// ---- Sequence/ST_SequenceInfo.TcDUT
{attribute 'enable_dynamic_creation'}
TYPE ST_SequenceInfo :
STRUCT
	nSequId 		: UDINT;			//4 Byte
	nStepNr 		: UINT;				//2 Byte
	eSequenceState	: E_SequenceState;	//1 Byte
	eStepState		: E_StepState;		//1 Byte
	nInfo			: DINT;				//4 Byte
END_STRUCT
END_TYPE

// ---- Sequence/ST_Step.TcDUT
{attribute 'enable_dynamic_creation'}
TYPE ST_Step :
STRUCT
	nStepNr				: UINT;	
	bStop				: BOOL;
	tDelay				: TIME;
	nTimerId			: USINT;
	eState 				: E_StepState;
	stActionData		: ST_ActionData;
	nActionId			: UINT;
	pCondi				: POINTER TO FB_CondiBase;
	aFollower			: ARRAY[0..9] OF UINT;
	bFollowerInQueue	: BOOL;	//Follwoer wurden in ProcessingQueue eingetragen
	bHasForerunner		: BOOL; //Hat einen Vorgänger (PreStep oder SpecStep) auf den gewartet wird
	bActionResultIsValid: BOOL;
	nActionResult		: DINT;
	nInfo				: DINT;
	bInfoChanged		: BOOL; //wird gesetzt, sobald sich der State oder nInfo ändert
END_STRUCT
END_TYPE

// ---- Configuration/GVL_ObjectArrays.TcGVL
{attribute 'contextName':='PlcTask'}
VAR_GLOBAL
	//Instanzierung der Objekte, sollten vom jeweiligem Objekttyp die Anzahl geändert werden müssen
	//dann die jeweilige Constante cMax....... ändern
	
	//MultiZ-Tools
	afbMzHead 			: ARRAY[1..cMaxMzHeads] OF FB_MzHead;				//MultiZ-Kopf - Anzahl bei 2 Ebenenplotter auf 2 Stück erhöhen
	afbPiezoPip 		: ARRAY[1..cMaxPiezoPips] OF FB_PiezoPip;			//Piezopipetten - Anzahl kann theoretisch auf 7 erhöht werden (pro Z-Scheibe 1 Pipette)
	afbPassivPip		: ARRAY[1..cMaxPassivPips] OF FB_PassivPip;			//Passivpipetten - Anzahl kann theoretisch auf 7 erhöht werden (pro Z-Scheibe 1 Pipette)
	afbPowderPip 		: ARRAY[1..cMaxPowderPips] OF FB_PowderPip;			//Pulverpipette
	afbMultiCartHolder	: ARRAY[1..cMaxMultiCartHolder] OF FB_MultiCartHolder;	//ehemals Corshell-Dispenser
	afbHybridDispenser	: ARRAY[1..cMaxHybridDispenser] OF FB_HybridDispenser;//
	afbCartDisp			: ARRAY[1..cMaxCartDisp] OF FB_CartDispenser;		//Kartuschen-Dispenser
	afbCartDispStirrer	: ARRAY[1..cMaxCartDispStirrer] OF FB_CartDispStirrer;	//Kartuschen-Dispenser mit Rührer
	afbCartHolder		: ARRAY[1..cMaxCartHolder] OF FB_CartHolder;		//Kartuschen-Halter
	afbCamera			: ARRAY[1..cMaxCameras] OF FB_Camera;				//Kamera oder Mikroskop oder Scanner
	afbZLevelSensor		: ARRAY[1..cMaxZLevelSensors] OF FB_ZLevelSensor;	//Z-Levelsensor
	afbStampSupport		: ARRAY[1..cMaxStampSupports] OF FB_StampSupport;	//Stempelkopf/Support
	afbDeloDot			: ARRAY[1..cMaxDeloDots] OF FB_DeloDot;				//DeloDot
	afbExposure			: ARRAY[1..cMaxExposure] OF FB_Exposure;			//Belichtung
	afbTriplePip		: ARRAY[1..cMaxTriplePip] OF FB_TriplePip;			//TriplePipette
	afbFlipTubeHandler	: ARRAY[1..cMaxFlipTubeHandler] OF FB_FlipTubeHandler;
	afbLuer				: ARRAY[1..cMaxLuer] OF FB_Luer;					
	afbVacuumHandler	: ARRAY[1..cMaxLuer] OF FB_VacuumHandler;
	afbSinglePiezoHolder: ARRAY[1..cMaxSinglePiezoHolder] OF FB_SingelPiezoHolder;
	afbTwinPiezoHolder	: ARRAY[1..cMaxTwinPiezoHolder] OF FB_TwinPiezoHolder;
	afbSolenoidPip		: ARRAY[1..cMaxSolenoidPip] OF FB_SolenoidPip;
	afbExtruder			: ARRAY[1..cMaxExtruder] OF FB_Extruder;
	afbpHElectrode		: ARRAY[1..cMaxpHElectrodes] OF FB_pHElectrode;
	afbTitrationTool	: ARRAY[1..cMaxTitrationTools] OF FB_TitrationTool;
	afbTwinExtruder		: ARRAY[1..cMaxTwinExtruder] OF FB_TwinExtruder;
	afbVermesDisp		: ARRAY[1..cMaxVermesDisp] OF FB_VermesDisp;
	afbDummyTool		: ARRAY[1..cMaxDummyTools] OF FB_DummyTool;	//Universelles Tool, welches außer den Move-Actions keine speziellen Funktionalitäten hat
	afbGripper			: ARRAY[1..cMaxGripper] OF FB_Gripper;
	afbPickPlacePip		: ARRAY[1..cMaxPickPlacePip] OF FB_PickPlacePip;
	
	//passive Targets
	afbWorkplate		: ARRAY[1..cMaxWorkplates] OF FB_Workplate;			//repräsentiert die gesamte Arbeitsfläche (Root) und kann nur 1x vorhanden sein
	afbSpotArray		: ARRAY[1..cMaxSpotArrays] OF FB_SpotArray;			//SpotArray
	afbDryPad			: ARRAY[1..cMaxDrayPads] OF FB_DryPad;				//Trockenpad
	afbSeptumWaste		: ARRAY[1..cMaxSeptumWaste] OF FB_SeptumWaste;		//SeptumWaste
	
	afbStampMagazine	: ARRAY[1..cMaxStampMagazines] OF FB_StampMagazine;	//Stempelmagazin
	afbSpotPattern		: ARRAY[1..cMaxSpotPatterns] OF FB_SpotPattern;		//Spotpattern
	afbNeedleRack		: ARRAY[1..cMaxNeedleRack] OF FB_NeedleRack;		//NeedleRack
	afbTipRack			: ARRAY[1..cMaxTipRack] OF FB_TipRack;				//TipRack
	afbFlipTubeRack		: ARRAY[1..cMaxFlipTubeRack] OF FB_FlipTubeRack;	//FlipTubeRack
	afbSeptumRack		: ARRAY[1..cMaxSeptumRack] OF FB_SeptumRack;		//SeptumRack
	afbVialRack			: ARRAY[1..cMaxVialRack] OF FB_VialRack;			//VialRack
	afbPortRack			: ARRAY[1..cMaxPortRack] OF FB_PortRack;			//PortRack
	afbpHElectrodeCapRack : ARRAY[1..cMaxpHElectrodeCapRack] OF FB_pHElectrodeCapRack;	//Rack für Konditionierungsgefäß pH-Elektrode
	afbTipCleanerGen2	: ARRAY[1..cMaxTipCleanerGen2] OF FB_TipCleanerGen2;
	
	//aktive Targets
	afbWashStation		: ARRAY[1..cMaxWashStations] OF FB_WashStation;		//Waschstation
	afbTipCleaner		: ARRAY[1..cMaxTipCleaners] OF FB_TipCleaner;		//Tip-Reinigung
	afbTipCalibrator	: ARRAY[1..cMaxTipCalibrators] OF FB_TipCalibrator;	//Tip-Kalibrierung
	afbStroboscope		: ARRAY[1..cMaxStroboscopes] OF FB_Stroboscope;		//Stroboskop
	afbMtpHolder		: ARRAY[1..cMaxMtpHolders] OF FB_MtpHolder;			//Mikrotiterplattenhalter, kann heizen oder kühlen
	afbSubstHolder		: ARRAY[1..cMaxSubstHolders] OF FB_SubstHolder;		//Substrathalter, kann heizen oder kühlen
	{IF defined(Unistat)}
	afbSubstHolderUnistat: ARRAY[1..cMaxSubstHolderUnistat] OF FB_SubstHolderUnistat;		//Substrathalter mit Huber Unistat 405
	{END_IF}
	afbInkStation		: ARRAY[1..cMaxInkStations] OF FB_InkStation;		//Lackschleuder für µCP
	afbPowderStation	: ARRAY[1..cMaxPowderStations] OF FB_PowderStation;	//Pulvervorrat für Pulverpipette
	afbReactor			: ARRAY[1..cMaxReactors] OF FB_Reactor;				//Reaktor
	afbLiquidReserve	: ARRAY[1..cMaxLiquidReserve] OF FB_LiquidReserve;	//LiquidReserve
	afbHighVoltTray		: ARRAY[1..cMaxHighVoltTray] OF FB_HighVoltTray;	//Hochspannungstablett für MES
	afbWorkplateCamera	: ARRAY[1..cMaxWorkplateCameras] OF FB_WorkplateCamera;
	afbCustomUnitType1	: ARRAY[1..cMaxCustomUnitTyp1] OF FB_CustomUnitType1;
	afbCustomUnitType2	: ARRAY[1..cMaxCustomUnitTyp2] OF FB_CustomUnitType2;
	afbTrayTransporter	: ARRAY[1..cMaxTrayTransporter] OF FB_TrayTransporter;
	
	//sonstige Devices
	afbDiluter			: ARRAY[1..cMaxDiluters] OF FB_Diluter;				//Spritzenpumpen
	afbDiluter3Inputs	: ARRAY[1..cMaxDiluters3Inputs] OF FB_Diluter3Inputs;
	afbStacker			: ARRAY[1..cMaxStacker] OF FB_Stacker;
	

	////////////////////////////////////////////////////////////////////////////////////////////////////////////////////////////////////////	
END_VAR

// ---- Configuration/GVL_ObjectConstants.TcGVL
VAR_GLOBAL CONSTANT
	//Legt die Anzahl der Instanzen der verschiedenen Objekt-Fbs fest.
	//Begrenzt die maximale Anzahl konfigurierbarer Objekt-Typen. 
	//MultiZ-Tools
	{IF defined (TwoHeads)}
	cMaxMzHeads			: USINT := 2;
	{ELSE}
	cMaxMzHeads			: USINT := 1;
	{END_IF}
	cMaxPickPlacePip	: UINT := 2;
	cMaxPiezoPips		: UINT := 4;
	cMaxPassivPips		: UINT := 8;
	cMaxPowderPips		: UINT := 1;
	cMaxMultiCartHolder	: UINT := 1;
	cMaxHybridDispenser	: UINT := 1;
	cMaxCartDisp		: UINT := 4;
	cMaxCartDispStirrer	: UINT := 1;
	cMaxCartHolder		: UINT := 6;
	cMaxCameras			: UINT := 6;
	cMaxZLevelSensors	: UINT := 2;
	cMaxStampSupports	: UINT := 1;
	cMaxDeloDots		: UINT := 1;
	cMaxExposure		: UINT := 4;
	cMaxTriplePip		: UINT := 2;
	cMaxFlipTubeHandler	: UINT := 1;
	cMaxLuer			: UINT := 6;
	cMaxVacuumHandler	: UINT := 2;
	cMaxSinglePiezoHolder: UINT := 4;
	cMaxTwinPiezoHolder	: UINT := 1;
	cMaxSolenoidPip		: UINT := 1;
	cMaxExtruder		: UINT := 4;
	cMaxpHElectrodes	: UINT := 1;
	cMaxTitrationTools	: UINT := 3;
	cMaxTwinExtruder	: UINT := 1;
	cMaxVermesDisp		: UINT := 1;
	cMaxDummyTools		: UINT := 7;
	cMaxGripper			: UINT := 1;
	
	//passive Targets
	cMaxWorkplates		: UINT := 1;
	cMaxSpotArrays		: UINT := 50;
	cMaxDrayPads		: UINT := 3;
	cMaxStampMagazines	: UINT := 1;
	cMaxSpotPatterns	: UINT := 10;
	cMaxSeptumWaste		: UINT := 1;
	cMaxNeedleRack		: UINT := 3;
	cMaxTipRack			: UINT := 2;
	cMaxFlipTubeRack	: UINT := 3;
	cMaxSeptumRack		: UINT := 1;
	cMaxVialRack		: UINT := 3;
	cMaxPortRack		: UINT := 1;
	cMaxpHElectrodeCapRack: UINT := 1;
	cMaxTipCleanerGen2	: UINT := 2;
	
	//aktive Targets
	cMaxWashStations	: UINT := 2;
	cMaxTipCleaners		: UINT := 1;
	cMaxTipCalibrators	: UINT := 1;
	cMaxStroboscopes	: UINT := 1;
	cMaxMtpHolders		: UINT := 3;
	cMaxSubstHolders	: UINT := 2;
	cMaxSubstHolderUnistat	: UINT := 1;
	cMaxInkStations		: UINT := 1;
	cMaxPowderStations	: UINT := 1;
	cMaxReactors		: UINT := 1;
	cMaxLiquidReserve	: UINT := 1;
	cMaxHighVoltTray	: UINT := 1;
	cMaxWorkplateCameras: UINT := 1;
	cMaxCustomUnitTyp1	: UINT := 2;
	cMaxCustomUnitTyp2	: UINT := 1;
	cMaxTrayTransporter : UINT := 1;
	
	//sonstige Devices
	cMaxDiluters		: UINT := 8;
	cMaxDiluters3Inputs	: UINT := 2;
	cMaxStacker			: UINT := 1;
	
	//!!!!!!!!!!!!!!!!!!!!!!!!!!!!!!!!!!!!!!!!!!!!!!!!!!!!!!!!!!!!!!!!!!!!!!!!!!!!!!!!!!!!!!!!!!!!!!!
	//Achtung, unbedingt cMaxObjects anpassen - muss "mindestens" die Summe aller cMax..... ergeben
	cMaxObjects			: UINT := 1000;
	
	//Achtung, unbedingt cMaxDevices anpassen - muss "mindestens" die Summe aller cMax.....  
	//von MultiZ-Tools + aktive Targets + sonstige Devices ergeben 
	cMaxDevices			: UINT := 30;

END_VAR

// ---- Configuration/GVL_ObjMgmt.TcGVL
VAR_GLOBAL
	fbConfiguration		: FB_Configuration;
	fbObjectDirectory 	: FB_ObjectDirectory;
	nObjPropChangeCnt	: USINT;
END_VAR

// ---- GVLs/GVL_Hardware.TcGVL
{attribute 'contextName':='PlcTask'}
VAR_GLOBAL CONSTANT
	//Definition der Hardwarecomponenten
	{define MtpHeater}
	{IF defined(MtpHeater)}
	cNoOfMtpHeaters	: USINT := 1;
	cNodeIdMtpHeater1 : USINT := 10;
	{END_IF}
	
	{define SubstHeater}
	{IF defined(SubstHeater)}
	cNoOfSubstHeaters : USINT := 1;
	cNodeIdSubstHeater1 : USINT := 12;
	{END_IF}

	//{define Reactor}
	{IF defined(Reactor)}
	cNoOfReactDrives : USINT := 1;
	cNodeIdReactDrive1	: USINT := 4;
	cNoOfReactHeaters : USINT := 1;
	cNodeIdReactHeater1	: USINT := 5;
	{END_IF}
	
	//{define BottleRack}
	{IF defined(BottleRack)}
	cNoOfBottleRacks : USINT := 1;
	cNodeIdBottleRack1 : USINT := 20;
	{END_IF}
	
	{define IOExpander}
	{IF defined(IOExpander)}
	cNoOfIOExpanders : USINT := 1;
	cNodeIdIOExpander1 : USINT := 16;
	{END_IF}
	
	//{define TripleTrigger}
	{IF defined(TripleTrigger)}
	cNoOfTripleTriggers : USINT := 1;
	cNodeIdTripleTrigger1 : USINT := 14;
	{END_IF}
	
	//{define PowderStation}
	{IF defined(PowderStation)}
	cNoOfPowderStations : USINT := 1;
	cNodeIdPowderStation1 : USINT := 24;
	{END_IF}
	
	//{define InkStation}
	{IF defined(InkStation)}
	cNoOfInkStatSpinDrives 		: USINT := 1;
	cNodeIdInkStatSpinDrive1	: USINT := 32;
	cNoOfInkStatCoverDrives 	: USINT := 1;
	cNodeIdInkStatCoverDrive1	: USINT := 33;
	{END_IF}
	
	{define MultiPurpIO}
	{IF defined(MultiPurpIO)}
	cNoOfMultiPurpIO			: USINT := 1;
	cNodeIdMultiPurpIO			: USINT := 25;
	{END_IF}
	
	cNoOfLiquidBottles 	: USINT := 1;
	cNoOfWasteBottles 	: USINT := 1;
	cNoOfPneuChannels	: USINT := 4;
	cNoOfPumps			: USINT := 9; //höchste Pumpennummer
	cNoOfGearPumps		: USINT := 4; //hochste Nummer Zahnradpumpen
	cNoOfValves			: USINT := 14;//höchste Ventilnummer
	cNoOfDiluters		: USINT	:= 8;
	
	cLiquidBottleNrPCV	: USINT := 1;
	
END_VAR

VAR_GLOBAL
	
	stPlcInfo			: ST_PlcInfo;	//Information über Seriennummer und Versionen der Plc
	
	//CAN-Nodes
	aCanNodes				: ARRAY[1..126] OF BOOL;
	
	//Settings
	fbSettings 				: FB_Settings;
	
	fbCANOpenHwModuleList	: FB_HwModuleList;	//alle GeSim CANopen-Module
	
	//Diluter	
	aFbDiluterRef			: ARRAY[1..cNoOfDiluters] OF FB_HwRefDiluter;
	
	//MultiZ-Module
	aFbMultiZRef			: ARRAY[1..cMaxMzHeads] OF FB_MultiZRef;	//Gerätereferenz zu MultiZ 1 (2)
	fbMultiZRefList			: FB_HwModuleList;
	
	{IF defined(MtpHeater)}
	aFbMtpHeatRef			: ARRAY[1..cNoOfMtpHeaters] OF FB_HwRef4ChHeater;
	{END_IF}
	
	{IF defined(SubstHeater)}
	aFbSubstHeatRef			: ARRAY[1..cNoOfSubstHeaters] OF FB_HwRef4ChHeater;
	{END_IF}	

	{IF defined(Reactor)}
	aFbReactDriveRef		: ARRAY[1..cNoOfReactDrives] OF FB_HwRefReactDrive;
	aFbReactHeatRef			: ARRAY[1..cNoOfReactHeaters] OF FB_HwRefReactHeater;
	{END_IF}
	
	{IF defined(BottleRack)}
	aFbBottleRackRef		: ARRAY[1..cNoOfBottleRacks] OF FB_HwRefBottleRack;
	{END_IF}
	
	{IF defined(IOExpander)}
	aFbIOExpanderRef		: ARRAY[1..cNoOfIOExpanders] OF FB_HwRefIOExpander;
	{END_IF}
	
	{IF defined(TripleTrigger)}
	aFbTripleTriggerRef		: ARRAY[1..cNoOfTripleTriggers] OF FB_HwRefTripleTrigger;
	{END_IF}
	
	{IF defined(PowderStation)}
	aFbPowderStatRef		: ARRAY[1..cNoOfPowderStations] OF FB_HwRefPowderStat;
	{END_IF}
	
	{IF defined(InkStation)}
	aFbInkStatDrvSpinRef	: ARRAY[1..cNoOfInkStatSpinDrives] OF FB_HwRefInkStatDriveSpin;
	aFbInkStatDrvCoverRef	: ARRAY[1..cNoOfInkStatCoverDrives] OF FB_HwRefInkStatDriveCover;
	{END_IF}
	
	//Muss in Compilerdefinitionen definiert werden
	{IF defined(TrayTransporterL)}
	fbHwRefTrayLock			: FB_HwRefTrayLock;
	fbHwRefTrayTransSlider 	: FB_HwRefNanotecPD;
	fbHwRefDrivingPinLeft	: FB_HwRefTMCM1140(bSetDigiOut0:= FALSE, bSetDigiOut1:= TRUE,
											eLimitSwitchLeftConfig := E_TMCM_SwitchConfig.Deactivated,
											eLimitSwitchRightConfig := E_TMCM_SwitchConfig.Deactivated,
											eHomeSwitchConfig := E_TMCM_SwitchConfig.Inverted,
											eHomingMethode := E_TMCM_HomingMethode.SearchNegHomeSwitch,
											nMicrostepResol := 64, nPulseDivisor := 2, nFullStepRevo := 200);
	{ELSIF defined(TrayTransporterR)}
	fbHwRefTrayLock			: FB_HwRefTrayLock;
	fbHwRefTrayTransSlider 	: FB_HwRefNanotecPD;
	fbHwRefDrivingPinRight	: FB_HwRefTMCM1140(bSetDigiOut0:= FALSE, bSetDigiOut1:= TRUE,
											eLimitSwitchLeftConfig := E_TMCM_SwitchConfig.Deactivated,
											eLimitSwitchRightConfig := E_TMCM_SwitchConfig.Deactivated,
											eHomeSwitchConfig := E_TMCM_SwitchConfig.Inverted,
											eHomingMethode := E_TMCM_HomingMethode.SearchNegHomeSwitch,
											nMicrostepResol := 64, nPulseDivisor := 2, nFullStepRevo := 200);
	{ELSIF defined(TrayTransporterLR)}
	fbHwRefTrayLock			: FB_HwRefTrayLock;
	fbHwRefTrayTransSlider  : FB_HwRefNanotecPD;
	fbHwRefDrivingPinLeft	: FB_HwRefTMCM1140(bSetDigiOut0:= FALSE, bSetDigiOut1:= TRUE,
											eLimitSwitchLeftConfig := E_TMCM_SwitchConfig.Deactivated,
											eLimitSwitchRightConfig := E_TMCM_SwitchConfig.Deactivated,
											eHomeSwitchConfig := E_TMCM_SwitchConfig.Inverted,
											eHomingMethode := E_TMCM_HomingMethode.SearchNegHomeSwitch,
											nMicrostepResol := 64, nPulseDivisor := 2, nFullStepRevo := 200);
	fbHwRefDrivingPinRight	: FB_HwRefTMCM1140(bSetDigiOut0:= FALSE, bSetDigiOut1:= TRUE,
											eLimitSwitchLeftConfig := E_TMCM_SwitchConfig.Deactivated,
											eLimitSwitchRightConfig := E_TMCM_SwitchConfig.Deactivated,
											eHomeSwitchConfig := E_TMCM_SwitchConfig.Inverted,
											eHomingMethode := E_TMCM_HomingMethode.SearchNegHomeSwitch,
											nMicrostepResol := 64, nPulseDivisor := 2, nFullStepRevo := 200);
	{END_IF}
	
	//Der jeweils erste Parameter muss mit der EtherCAT Addr der zugeordneten Klemme übereinstimmen.
	{IF defined (Stacker)}
	fbHwRefSpinDrive	: FB_HwRefEL70xxDriveExtEncoder(1011, E_EL70xx_StartType.SetCalibration, E_EL70xx_EncoderType.ExternSingleturnAbs, 262144); //Encoder mit 18bit Auflösung);
	fbHwRefLiftDrive	: FB_HwRefEL70xxDrive(1013, E_EL70xx_StartType.CaliHwSync);
	fbHwRefTrayStop		: FB_HwRefEL70xxDrive(1014, E_EL70xx_StartType.CaliPlcCam);
	{END_IF}
	
	//TipCleaner
	stTipCleanerRef			: ST_TipCleanerRef;
	
	//TipCalibrator
	stTipCalibrator			: ST_TipCalibrator;
	
	//FBox
	aValves					: ARRAY[1..cNoOfValves] OF FB_Valve;
	aPumps					: ARRAY[1..cNoOfPumps] OF FB_Pump;
	aFbGearPumps			: ARRAY[1..cNoOfGearPumps] OF FB_GearPump;
	aSensSysLiquidBottle	AT %I* : ARRAY[1..cNoOfLiquidBottles] OF BOOL;	
	aSensWasteBottle		AT %I* : ARRAY[1..cNoOfWasteBottles] OF BOOL;
	
	{IF defined(MultiPurpIO)}
	aFbHwRefMultiPurpIO		: ARRAY[1..cNoOfMultiPurpIO] OF FB_HwRefMultiPurpIO;
	{END_IF}
	
	//Pneumatik-Kanäle
	aFbPneuChannel			: ARRAY[1..cNoOfPneuChannels] OF FB_PneuChannelRef;
	
	fbPCV					: FB_PCV;
	
	//Hochspannungsquelle	
	{define HighVoltSupply}
	{IF defined(HighVoltSupply)}
	fbHighVoltSupplyRef		: FB_HighVoltSupply;
	{END_IF}

	{IF defined(FDM1)}
	//Referenz zur Pulse Train Klemme für FDM-Head von STEPCRAFT
	stPTOStepperRef			: ST_PTOStepperRef;
	fbFDM_EL2521Ref			: FB_FDM_EL2521_Ref(ADR(stPTOStepperRef));
	{END_IF}
	
	{IF defined(FDM2)}
	fbHwRefFDM_TMCM	: FB_HwRefTMCM1140(bSetDigiOut0:= TRUE, bSetDigiOut1:= FALSE,
									eLimitSwitchLeftConfig := E_TMCM_SwitchConfig.Deactivated,
									eLimitSwitchRightConfig := E_TMCM_SwitchConfig.Deactivated,
									eHomeSwitchConfig := E_TMCM_SwitchConfig.Deactivated,
									eHomingMethode := E_TMCM_HomingMethode.NoHoming,
									nMicrostepResol := 256, nFullStepRevo := 200, nRampDivisor:= 7, nPulseDivisor := 2);
	fbEndlessExtrTMCMRef	: FB_EndlessExtruderTMCM_Ref(ADR(fbHwRefFDM_TMCM));									
	{END_IF}
	
	{IF defined(Pure1)}
	fbHwRefTMCM_Pure1	: FB_HwRefTMCM1140(bSetDigiOut0:= TRUE, bSetDigiOut1:= FALSE,
									eLimitSwitchLeftConfig := E_TMCM_SwitchConfig.Deactivated,
									eLimitSwitchRightConfig := E_TMCM_SwitchConfig.Deactivated,
									eHomeSwitchConfig := E_TMCM_SwitchConfig.Deactivated,
									eHomingMethode := E_TMCM_HomingMethode.NoHoming,
									nMicrostepResol := 8, nFullStepRevo := 24, nRampDivisor:= 7, nPulseDivisor := 2);
	fbEndlessExtrTMCMRef_Pure1	: FB_EndlessExtruderTMCM_Ref(ADR(fbHwRefTMCM_Pure1));									
	{END_IF}
	
	{IF defined(Pure2)}
	fbHwRefTMCM_Pure2	: FB_HwRefTMCM1140(bSetDigiOut0:= TRUE, bSetDigiOut1:= FALSE,
									eLimitSwitchLeftConfig := E_TMCM_SwitchConfig.Deactivated,
									eLimitSwitchRightConfig := E_TMCM_SwitchConfig.Deactivated,
									eHomeSwitchConfig := E_TMCM_SwitchConfig.Deactivated,
									eHomingMethode := E_TMCM_HomingMethode.NoHoming,
									nMicrostepResol := 8, nFullStepRevo := 24, nRampDivisor:= 7, nPulseDivisor := 2);
	fbEndlessExtrTMCMRef_Pure2	: FB_EndlessExtruderTMCM_Ref(ADR(fbHwRefTMCM_Pure2));									
	{END_IF}
	
	{IF defined(Pure3)}
	fbHwRefTMCM_Pure3	: FB_HwRefTMCM1140(bSetDigiOut0:= TRUE, bSetDigiOut1:= FALSE,
									eLimitSwitchLeftConfig := E_TMCM_SwitchConfig.Deactivated,
									eLimitSwitchRightConfig := E_TMCM_SwitchConfig.Deactivated,
									eHomeSwitchConfig := E_TMCM_SwitchConfig.Deactivated,
									eHomingMethode := E_TMCM_HomingMethode.NoHoming,
									nMicrostepResol := 8, nFullStepRevo := 24, nRampDivisor:= 7, nPulseDivisor := 2);
	fbEndlessExtrTMCMRef_Pure3	: FB_EndlessExtruderTMCM_Ref(ADR(fbHwRefTMCM_Pure3));									
	{END_IF}
	
	{IF defined(SCREWEXTR1)}
	fbHwRefScrewExtr_TMCM	: FB_HwRefTMCM1140_Gen2(bSetDigiOut0:= FALSE, bSetDigiOut1:= FALSE,
									eLimitSwitchLeftConfig := E_TMCM_SwitchConfig.Deactivated,
									eLimitSwitchRightConfig := E_TMCM_SwitchConfig.Deactivated,
									eHomeSwitchConfig := E_TMCM_SwitchConfig.Deactivated,
									eHomingMethode := E_TMCM_HomingMethode.NoHoming,
									nMicrostepResol := 256, nPulseDivisor := 2, nFullStepRevo := 200);
	{END_IF}
	
	//Referenz zum Huber Unistat
	{IF defined(Unistat)}
	fbUnistatRef			: FB_HwRefUnistat(GVL_RS232.fbSerialPortUnistat);
	{END_IF}
	
	//Safety
	fbSafety				: FB_Safety;
	fbSafetyPseudo			: FB_SafetyPseudo;		//nur für ein spezielles Gerät (IWS)
	fbSafetyBase			: FB_SafetyBase;
	pFbSafety				: POINTER TO FB_SafetyBase; //dieser Zeiger verweist auf die eigentliche Safety Instanz, welche in "ScanHwModules" diesem
													//Zeiger in Abhängigkeit von der Hardware zugeordnet wird und dann entsprechend in "PerformHardware"
													//aufgerufen wird
													
	{IF defined(Stacker)}
	fbSafetyStacker 		: FB_SafetyStacker;
	fbSignalLightStacker	: FB_SignalLight;	
	{END_IF}
													
	fbStopButton	: FB_HwRefStopButton;
	
	fbSignalLight	: FB_SignalLight;
	
	fbPlcTriggerOut	: FB_TriggerOut;
	
	fbMultiZDigiOut : FB_TriggerOut;
	
	fbMultiZPWM		: FB_MultiZPWM;

	//XY-Antriebe
	//NC-Achsenreferenzen (mit Ec-Slaves verknüpfen und NC-Achsen zuweisen
	AxisRefX1		: Tc2_MC2.AXIS_REF;
	AxisRefX2		: Tc2_MC2.AXIS_REF;	//derzeit nur Plattform C
	AxisRefY1		: Tc2_MC2.AXIS_REF;	//bei Plattform D unten
	AxisRefY2		: Tc2_MC2.AXIS_REF; //bei Plattform D oben

	AxisRefQ1		: Tc2_MC2.AXIS_REF;	//Virtuelle Achse(Z) für GCode
	
	//Linmot-Achsenreferenzen (nur für Antriebe C1100-EC-XC)
	lmAxisRefX		: Tc3_LinMot.tstLM_Axis;
	lmAxisRefY1		: Tc3_LinMot.tstLM_Axis; //untere Achse
	lmAxisRefY2		: Tc3_LinMot.tstLM_Axis; //obere Achse
	
	
	fbX1DriveLmtDS	: FB_XYDrive_Lmt_DS(pNCAxisRef:= ADR(AxisRefX1), eXYOrientation:= E_XYOrientation.X);
	fbY1DriveLmtDS	: FB_XYDrive_Lmt_DS(pNCAxisRef:= ADR(AxisRefY1), eXYOrientation:= E_XYOrientation.Y);
	fbY2DriveLmtDS	: FB_XYDrive_Lmt_DS(pNCAxisRef:= ADR(AxisRefY2), eXYOrientation:= E_XYOrientation.Y);
	
	fbX1DriveLmtEC	: FB_XYDrive_Lmt_EC(pAxisRef:= ADR(lmAxisRefX), eXYOrientation:= E_XYOrientation.X);
	fbY1DriveLmtEC	: FB_XYDrive_Lmt_EC(pAxisRef:= ADR(lmAxisRefY1),eXYOrientation:= E_XYOrientation.Y);
	fbY2DriveLmtEC	: FB_XYDrive_Lmt_EC(pAxisRef:= ADR(lmAxisRefY2),eXYOrientation:= E_XYOrientation.Y);	
	
	fbXDriveBeck	: FB_XYDrive_Beck_Twin(pNCAxisRefMaster:= ADR(AxisRefX1), pNCAxisRefSlave:= ADR(AxisRefX2), eXYOrientation:= E_XYOrientation.X);
	fbYDriveBeck	: FB_XYDrive_Beck(pNCAxisRefMaster:= ADR(AxisRefY1), eXYOrientation:= E_XYOrientation.Y);
	
	fbXYDriveList 	: FB_HwModuleList;	//wird in Prog "ScanHwModules" gefüllt

END_VAR

// ---- GVLs/GVL_RS232.TcGVL
{attribute 'qualified_only'}
{attribute 'contextName':='ComTask'}
VAR_GLOBAL CONSTANT
	{IF defined(Unistat) AND defined(Diluter)}
	cNoOfSerialPorts 	: USINT := 2;
	{ELSE}
	cNoOfSerialPorts 	: USINT := 1;
	{END_IF} 	
END_VAR

VAR_GLOBAL
	{IF defined(CX5010) AND defined(Unistat) AND defined(Diluter)}
	fbSerialPortDiluter	: FB_SerialComPort_PC;
	fbSerialPortUnistat	: FB_SerialComPort_USB;
	aSerialPorts	: ARRAY[1..cNoOfSerialPorts] OF POINTER TO FB_SerialComPort_Base := [ADR(fbSerialPortDiluter), ADR(fbSerialPortUnistat)];
	{ELSIF defined(CX5010) OR defined(CX9020)}
	fbSerialPortDiluter	: FB_SerialComPort_PC;
	aSerialPorts	: ARRAY[1..cNoOfSerialPorts] OF POINTER TO FB_SerialComPort_Base := [ADR(fbSerialPortDiluter)];
	{ELSIF defined(C6015) AND defined(Unistat) AND defined(Diluter)} //kam bisher noch nicht vor
	fbSerialPortDiluter	: FB_SerialComPort_EL60xx;
	fbSerialPortUnistat	: FB_SerialComPort_USB;
	aSerialPorts	: ARRAY[1..cNoOfSerialPorts] OF POINTER TO FB_SerialComPort_Base := [ADR(fbSerialPortDiluter), ADR(fbSerialPortUnistat)];
	{ELSIF defined(C6015) AND defined(Unistat)}
	fbSerialPortUnistat	: FB_SerialComPort_USB;
	fbSerialPortDiluter	: FB_SerialComPort_Base; //nur als Dummy
	aSerialPorts	: ARRAY[1..cNoOfSerialPorts] OF POINTER TO FB_SerialComPort_Base := [ADR(fbSerialPortUnistat)];
	{ELSE}
	fbSerialPortDiluter	: FB_SerialComPort_USB;
	aSerialPorts	: ARRAY[1..cNoOfSerialPorts] OF POINTER TO FB_SerialComPort_Base := [ADR(fbSerialPortDiluter)];
	{END_IF}
END_VAR

// ---- GVLs/GVL_Sm.TcGVL
VAR_GLOBAL
	fbComplexAction		: FB_ComplexAction;
	
	//Variablen für Ads-Notifictaion
	aObjProcData		: ARRAY[1..(cMaxDevices + cMaxDrayPads)] OF ST_ObjectProcData;
	
	//aktuelle Werte der Pneu-Channels und der Interlocks
	aHardwProcData		: ARRAY[0..13] OF ST_HardwareProcData;

	//Variablen für Interaktive Kommunikation während der Abarbeitung von Actionen
	stInteractRequest	: ST_Interaction;
	stInterResponse		: ST_Interaction;
	
	timeStamp 			: T_FILETIME;//Locale Sytemzeit für ST_Error.TimeStamp
	//Errorstruktur
	stNotifyError		: ST_Error;
	fbErrorList			: FB_ErrorList;
	
	//Für Notification der aktuellen Sequenzabarbeitung
	fbSequenceList		: FB_SequenceList;	
	fbSequenceInfo		: FB_SequenceInfo;
	stSequenceInfo		: ST_SequenceInfo;
	
END_VAR

// ---- Hardware/MultiZ/GVL_MultiZObjects.TcGVL
VAR_GLOBAL CONSTANT
	cForceThrshld 				: ST_CANopenObject:= (nIndex:= 16#2006, nLength:= 2);
	cForcePos 					: ST_CANopenObject:= (nIndex:= 16#2007, nLength:= 4);
	cForceVelo 					: ST_CANopenObject:= (nIndex:= 16#2008, nLength:= 2);
	cCurrentPos 				: ST_CANopenObject:= (nIndex:= 16#2009, nLength:= 4);
	cGPInputMode 				: ST_CANopenObject:= (nIndex:= 16#2100, nLength:= 1);
	cAnaInTrigg 				: ST_CANopenObject:= (nIndex:= 16#2101, nLength:= 1);
	cAnaInLimit					: ST_CANopenObject:= (nIndex:= 16#2102, nLength:= 2);
	cAnaInDelta					: ST_CANopenObject:= (nIndex:= 16#2003, nLength:= 2);
	cPwmEnable 					: ST_CANopenObject:= (nIndex:= 16#2200, nLength:= 1);
	cPwmValue 					: ST_CANopenObject:= (nIndex:= 16#2201, nLength:= 2);
	cAnaOutEnable 				: ST_CANopenObject:= (nIndex:= 16#2200, nLength:= 2);
	cAnaOutValue				: ST_CANopenObject:= (nIndex:= 16#2201, nLength:= 2);
	cHardVersion 				: ST_CANopenObject:= (nIndex:= 16#1009, nLength:= 15);
	cSoftVersion 				: ST_CANopenObject:= (nIndex:= 16#100A, nLength:= 15);
	cTMCVersion 				: ST_CANopenObject:= (nIndex:= 16#2010, nLength:= 4);
	cZSensOffset 				: ST_CANopenObject:= (nIndex:= 16#2424, nLength:= 4);
	cToolEnable 				: ST_CANopenObject:= (nIndex:= 16#2400, nLength:= 1);
	cToolType 					: ST_CANopenObject:= (nIndex:= 16#2401, nLength:= 1);
	cHeaterExist 				: ST_CANopenObject:= (nIndex:= 16#2402, nLength:= 1);
	cTempSetPoint 				: ST_CANopenObject:= (nIndex:= 16#2410, nLength:= 2);
	cTempSetPoint2 				: ST_CANopenObject:= (nIndex:= 16#2412, nLength:= 2);
	cTempSetPoint3 				: ST_CANopenObject:= (nIndex:= 16#2414, nLength:= 2);
	cHeatingOn 					: ST_CANopenObject:= (nIndex:= 16#2404, nLength:= 1);
	cPiezoPeriod 				: ST_CANopenObject:= (nIndex:= 16#2420, nLength:= 2);
	cPiezoPulse 				: ST_CANopenObject:= (nIndex:= 16#2421, nLength:= 2);
	cPiezoDrops 				: ST_CANopenObject:= (nIndex:= 16#2422, nLength:= 2);
	cPiezoVoltage 				: ST_CANopenObject:= (nIndex:= 16#2423, nLength:= 2);
	cPiezoHoldVoltage 			: ST_CANopenObject:= (nIndex:= 16#2426, nLength:= 2);
	cPiezoPrePeakTime 			: ST_CANopenObject:= (nIndex:= 16#2425, nLength:= 2);
	cPiezoStrobTest				: ST_CANopenObject:= (nIndex:= 16#2300, nSubIndex:= 1, nLength:= 1);
	cPiezoCamDelay 				: ST_CANopenObject:= (nIndex:= 16#2300, nSubIndex:= 2, nLength:= 2);
	cPiezoStrobDelay			: ST_CANopenObject:= (nIndex:= 16#2300, nSubIndex:= 3, nLength:= 2);
	cPiezoStrobDelay2			: ST_CANopenObject:= (nIndex:= 16#2300, nSubIndex:= 4, nLength:= 2);
	cTriggerVersion				: ST_CANopenObject:= (nIndex:= 16#2300, nSubIndex:= 5, nLength:= 1);
	cPiezoStrobDroplistActive	: ST_CANopenObject:= (nIndex:= 16#2301, nSubIndex:= 1, nLength:= 1);
	cPiezoStrobDroplist1_4		: ST_CANopenObject:= (nIndex:= 16#2301, nSubIndex:= 2, nLength:= 4);
	cPiezoStrobDroplist5_8		: ST_CANopenObject:= (nIndex:= 16#2301, nSubIndex:= 3, nLength:= 4);
	cPiezoStrobDroplist9_12		: ST_CANopenObject:= (nIndex:= 16#2301, nSubIndex:= 4, nLength:= 4);
	cPiezoStrobDroplist13_16	: ST_CANopenObject:= (nIndex:= 16#2301, nSubIndex:= 5, nLength:= 4);
	cRefPos						: ST_CANopenObject:= (nIndex:= 16#2011, nLength:= 4);
	cExtruderFeed				: ST_CANopenObject:= (nIndex:= 16#2430, nLength:= 2);
	cExtruderCompressFeed		: ST_CANopenObject:= (nIndex:= 16#2431, nLength:= 2);
	cExtruderRelaxFeed			: ST_CANopenObject:= (nIndex:= 16#2432, nLength:= 2);
	cExtruderDistance			: ST_CANopenObject:= (nIndex:= 16#2433, nLength:= 2);
	cExtruderCompressDistance	: ST_CANopenObject:= (nIndex:= 16#2434, nLength:= 2);
	cExtruderRelaxDistance		: ST_CANopenObject:= (nIndex:= 16#2435, nLength:= 2);
	cExtruderUnlockOffset		: ST_CANopenObject:= (nIndex:= 16#2437, nLength:= 4);
	cToolVersion				: ST_CANopenObject:= (nIndex:= 16#2406, nLength:= 1);
	
	
	cConfigFix					: ST_CANopenObject:= (nIndex:= 16#24FF, nSubIndex:= 1, nLength:= 1);
	cConfigCRC					: ST_CANopenObject:= (nIndex:= 16#24FF, nSubIndex:= 2, nLength:= 2);
	cuCPCtrl					: ST_CANopenObject:= (nIndex:= 16#2500, nSubIndex:= 1, nLength:= 1);
	cuCPMode					: ST_CANopenObject:= (nIndex:= 16#2500, nSubIndex:= 2, nLength:= 1);
	cuCPAngleSetpoint			: ST_CANopenObject:= (nIndex:= 16#2500, nSubIndex:= 3, nLength:= 2);
	cuCPSpinSpeed				: ST_CANopenObject:= (nIndex:= 16#2500, nSubIndex:= 6, nLength:= 4);
	cuCPLock					: ST_CANopenObject:= (nIndex:= 16#2500, nSubIndex:= 7, nLength:= 1);
	cuCPUnlockOffset			: ST_CANopenObject:= (nIndex:= 16#2500, nSubIndex:= 8, nLength:= 4);
	cuCPLight					: ST_CANopenObject:= (nIndex:= 16#2500, nSubIndex:= 9, nLength:= 1);
	
	cGlobError					: ST_CANopenObject:= (nIndex:= 16#5FFF, nSubIndex:= 8, nLength:= 1);
	cLastErrorState				: ST_CANopenObject:= (nIndex:= 16#5FFE, nSubIndex:= 0, nLength:= 4);
	
	cUpdateRequest				: ST_CANopenObject:= (nIndex:= 16#4000, nSubIndex:= 8, nLength:= 1);
	
	
	
END_VAR

// ---- Hardware/Trigger/GVL_HwRefIO.TcGVL
VAR_GLOBAL
	bTrigger1 AT %Q*: BOOL; //genutzt von Exposer oder StampSupport
	//bTrigger1 wird seid V2.0.17.27 nicht mehr genutzt
	//Es gibt dafür in GVL_Hardware: 
	//fbPlcTriggerOut	: FB_TriggerOut;
	//fbMultiZDigiOut 	: FB_TriggerOut;
	//fbMultiZPWM		: FB_MultiZPWM;
	bTrigger2 AT %Q*: BOOL;	//genutzt von M150/M151 (GCode)
END_VAR

// ---- Version/Global_Version.TcGVL
{attribute 'TcGenerated'}
{attribute 'no-analysis'}
{attribute 'linkalways'}
// This function has been automatically generated from the project information.
VAR_GLOBAL CONSTANT
	{attribute 'const_non_replaced'}
	stLibVersion_SPS_PlattformCD : ST_LibVersion := (iMajor := 2, iMinor := 0, iBuild := 18, iRevision := 19, nFlags := 0, sVersion := '2.0.18.19');
END_VAR

// ---- Objects/Interfaces/I_Dispenser.TcIO
INTERFACE I_Dispenser EXTENDS I_Device

METHOD M_DispenserPrepare : ERRORID
VAR_INPUT
END_VAR
END_METHOD

METHOD M_DispenserStart : ERRORID
VAR_INPUT
END_VAR
END_METHOD

METHOD M_DispenserStop : ERRORID
VAR_INPUT
END_VAR
END_METHOD

PROPERTY P_bError : BOOL
GET
END_GET
END_PROPERTY

PROPERTY P_eDispenserState : E_DispenserState
GET
END_GET
END_PROPERTY

PROPERTY P_nErrorId : ERRORID
GET
END_GET
END_PROPERTY

PROPERTY P_pObject : POINTER TO FB_Object
GET
END_GET
END_PROPERTY

END_INTERFACE

// ---- Objects/Interfaces/I_SlotTarget.TcIO
INTERFACE I_SlotTarget

METHOD M_GetSlot : POINTER TO FB_Slot
VAR_INPUT
	nSlotNr : UINT;
END_VAR
END_METHOD

METHOD M_GetSlotFromChild : POINTER TO FB_Slot
VAR_INPUT
	pObject : POINTER TO FB_Object;
END_VAR
END_METHOD

END_INTERFACE

// ---- Objects/Interfaces/I_Device.TcIO
INTERFACE I_Device

PROPERTY P_bBusy : BOOL
GET
END_GET
END_PROPERTY

METHOD M_GetProcData : DINT
VAR_INPUT
	eProcDataType : E_ProcDataType;
END_VAR
END_METHOD

PROPERTY P_bError : BOOL
GET
END_GET
END_PROPERTY

METHOD M_GetActionBusy : BOOL
VAR_INPUT
	eAction : E_Action;
END_VAR
END_METHOD

METHOD M_Stop : ERRORID
VAR_INPUT
END_VAR
END_METHOD

METHOD M_ExeAction : ERRORID
VAR_INPUT
	refActionData : REFERENCE TO ST_ActionData;
END_VAR
END_METHOD

PROPERTY P_pObject : POINTER TO FB_Object
GET
END_GET
END_PROPERTY

PROPERTY P_bCanceled : BOOL
GET
END_GET
END_PROPERTY

METHOD M_Reset
VAR_INPUT
END_VAR
END_METHOD

PROPERTY P_bStopAllOnError : BOOL
GET
END_GET
END_PROPERTY

PROPERTY P_bIsInit : BOOL
GET
END_GET
END_PROPERTY

METHOD M_CheckAction : ERRORID
VAR_INPUT
	refActionData 	: REFERENCE TO ST_ActionData;
	pCorrelObject	: POINTER TO FB_Object;
END_VAR
END_METHOD

METHOD M_CheckProcDataType : BOOL
VAR_INPUT
	eProcDataType : E_ProcDataType;
END_VAR
END_METHOD

METHOD M_CancelAction
VAR_INPUT
	eAction : E_Action;
END_VAR
END_METHOD

PROPERTY P_eCurrentState : E_MachineState
GET
END_GET
END_PROPERTY

PROPERTY P_nErrorId : ERRORID
GET
END_GET
END_PROPERTY

PROPERTY P_stError : ST_Error
GET
END_GET
END_PROPERTY

END_INTERFACE

// ---- Objects/Interfaces/I_TargetZSensor.TcIO
INTERFACE I_TargetZSensor

PROPERTY P_bSensor : BOOL
GET
END_GET
END_PROPERTY

END_INTERFACE

// ---- Objects/Interfaces/I_UsingDryPad.TcIO
INTERFACE I_UsingDryPad

PROPERTY P_tDryTime : TIME
GET
END_GET
END_PROPERTY

PROPERTY P_nDrypadArea : USINT
GET
END_GET
END_PROPERTY

END_INTERFACE

// ---- Hardware/CANInterfaceCom.TcPOU
{attribute 'contextName':='ComTask'}
PROGRAM CANInterfaceCom
VAR
	//Input
	nInTxCounter 		AT %I* : UINT;
	nInRxCounter 		AT %I* : UINT;
	nInCobId			AT %I* : UINT;
	aInData				AT %I* : ARRAY[0..7] OF USINT;
	//Output
	nOutTxCounter 		AT %Q* : UINT;
	nOutRxCounter 		AT %Q* : UINT;
	nOutNoOfTxMessages	AT %Q* : UINT := 1;
	nOutCobId			AT %Q* : UINT;
	aOutData			AT %Q* : ARRAY[0..7] OF USINT;
	nState				: USINT;
	bInit				: BOOL := TRUE;
	stCanInterfaceBuffer: ST_CANInterfaceBuffer;
END_VAR

IF bInit THEN
	F_CreateLinkedListHnd( ADR(stCanInterfaceBuffer.aNodes ), SIZEOF( stCanInterfaceBuffer.aNodes ), stCanInterfaceBuffer.hList );
	bInit := FALSE;
END_IF

IF stCanInterfaceBuffer.bExecute THEN
	IF nState = 0 THEN
		stCanInterfaceBuffer.bBusy := TRUE;
		nOutRxCounter := nInRxCounter;
		//CobId aus Identifier und Datenlänge bilden
		nOutCobId := SHL(stCanInterfaceBuffer.nTxIdent,5) OR stCanInterfaceBuffer.nTxDlc;
		aOutData := stCanInterfaceBuffer.aTxData;
		//durch inkrementieren durch nOutTxCounter wird gesendet
		nOutTxCounter := nOutTxCounter + 1;
		nState := 1;
	ELSIF nState = 1 THEN //auf Rx warten
		IF nInRxCounter <> nOutRxCounter THEN
			//Identifier und Datenlänge extrahieren
			stCanInterfaceBuffer.nRxIdent := SHR(nInCobId,5);
			stCanInterfaceBuffer.nRxDlc := UINT_TO_USINT(nInCobId) AND 16#0F;
			MEMSET(ADR(stCanInterfaceBuffer.aRxData),0,8);
			MEMCPY(ADR(stCanInterfaceBuffer.aRxData),ADR(aInData),stCanInterfaceBuffer.nRxDlc);
			//Empfang bestätigen
			nOutRxCounter := nInRxCounter;
			stCanInterfaceBuffer.bBusy := FALSE;
			nState := 80;
		END_IF
	END_IF
ELSE
	nState := 0;
END_IF

END_PROGRAM

// ---- Hardware/RS232/SerialBackCom.TcPOU
{attribute 'contextName':='ComTask'}
PROGRAM SerialBackCom
VAR
	i : USINT;
END_VAR

FOR i:= 1 TO GVL_RS232.cNoOfSerialPorts BY 1 DO
	IF GVL_RS232.aSerialPorts[i] > 0 THEN
		GVL_RS232.aSerialPorts[i]^();	
	END_IF
END_FOR

END_PROGRAM

// ---- FirmwUpdate/FirmwUpdate.TcPOU
PROGRAM FirmwUpdate
VAR_INPUT
	pFbCanNode : POINTER TO FB_CanNodeBase;
	bExecute	: BOOL;
END_VAR
VAR_OUTPUT
	bBusy : BOOL;
	bError : BOOL;
	nErrorId : ERRORID;
	stInfo : ST_FirmwUpdInfo;
END_VAR
VAR
	nStateAction			: UINT;
	nStateActionNext		: UINT;
	nStateActionTimeout		: UINT;
	fbSendCanMessage 		: FB_SendCanMessage(ADR(CANInterfaceCom.stCanInterfaceBuffer));
	fbS19File				: FB_S19File;
	aExpectedData			: ARRAY[0..7] OF USINT;
END_VAR

//0. File laden und verifizieren
//1. Check, ob Node da
//2. Node da? -> reset
//3. Connect so lange ausführen, bis positive Antwort
//4. Status abrufen
//5. Programm start
//6. Set_MTA
//7. Programm clear
//8. Alle Blöcke schreiben
//9. Programm Ende
//10. Programm Reset
IF bExecute THEN
	CASE nStateAction OF
		0:	//File laden
			IF pFbCanNode = 0 THEN
				nErrorId := E_ErrorIdHwGeneral.ERRORID_InvalidHwRef;
				nStateAction := 99;
				bError := TRUE;
				RETURN;
			END_IF
			stInfo.eActState := E_FirmwUpdState.LoadFile;
			stInfo.nBytesToWrite := 0;
			stInfo.nWrittenBytes := 0;
			bBusy := TRUE;
			{IF defined(WIN10)}
			fbS19File.A_OpenFile(sFileName:= 'C:\ftp\FirmwUpdate\FirmwUpdate.s19', bExecute:= TRUE);
			{ELSE}
			fbS19File.A_OpenFile(sFileName:= '\Hard Disk\ftp\FirmwUpdate\FirmwUpdate.s19', bExecute:= TRUE);
			{END_IF}
			IF NOT fbS19File.bBusy THEN
				IF fbS19File.bError THEN
					nErrorId := fbS19File.nErrorId;
					nStateAction := 99;
				ELSE
					//Node vorhanden?
					IF pFbCanNode^.P_bNodeEnabled AND pFbCanNode^.P_nNodeState = 0 THEN
						pFbCanNode^.P_bStopMonitor := TRUE;	//Überwachung des Node deaktivieren
						pFbCanNode^.M_ResetApp();
					END_IF
					nStateAction := 1;
				END_IF
				fbS19File.A_OpenFile(bExecute:= FALSE);
			END_IF
			
		1:	//CONNECT
			stInfo.eActState := E_FirmwUpdState.Connect;
			stInfo.nBytesToWrite := fbS19File.P_nBytesToWrite;
			fbSendCanMessage.aTxData[0] := 16#FF;	//XCP-Command: CONNECT
			fbSendCanMessage.aTxData[1] := 0;
			fbSendCanMessage.tTimeout := T#40MS;
			fbSendCanMessage.nTxLength := 2;
			nStateActionNext := 2;
			nStateActionTimeout := 1;
			nStateAction := 60;
			//Erwartete Antwort
			HEXSTR_TO_DATA('FF10000808000101',ADR(aExpectedData),8);
			
		2:	//GET_STATUS
			stInfo.eActState := E_FirmwUpdState.GetStatus;
			fbSendCanMessage.aTxData[0] := 16#FD;	//XCP-Command: GET_STATUS
			fbSendCanMessage.tTimeout := T#100MS;
			fbSendCanMessage.nTxLength := 1;
			nStateActionNext := 3;
			nStateActionTimeout := 99;
			nStateAction := 60;
			//Erwartete Antwort
			HEXSTR_TO_DATA('FF00000000000000',ADR(aExpectedData),8);
			
		3:	//PROGRAM_START
			stInfo.eActState := E_FirmwUpdState.ProgramStart;
			fbSendCanMessage.aTxData[0] := 16#D2;	//XCP-Command: PROGRAM_START
			fbSendCanMessage.tTimeout := T#100MS;
			fbSendCanMessage.nTxLength := 1;
			nStateActionNext := 4;
			nStateActionTimeout := 99;
			nStateAction := 60;
			//Erwartete Antwort
			HEXSTR_TO_DATA('FF00000800000000',ADR(aExpectedData),8);
			
		4:	//SET_MTA
			stInfo.eActState := E_FirmwUpdState.SetMTA;
			fbSendCanMessage.aTxData[0] := 16#F6;	//XCP-Command: SET_MTA
			fbS19File.M_GetStartAdress(ADR(fbSendCanMessage.aTxData[4])); //ab hier wird das Programm im nächsten Schritt gelöscht
			fbSendCanMessage.tTimeout := T#100MS;
			fbSendCanMessage.nTxLength := 8;
			nStateActionNext := 5;
			nStateActionTimeout := 99;
			nStateAction := 60;
			//Erwartete Antwort
			HEXSTR_TO_DATA('FF00000000000000',ADR(aExpectedData),8);
			
		5:	//PROGRAM_CLEAR - 
			stInfo.eActState := E_FirmwUpdState.ProgramClear;
			fbSendCanMessage.aTxData[0] := 16#D1;	//XCP-Command: PROGRAM_CLEAR
			fbS19File.M_GetNoOfTotalBytes(ADR(fbSendCanMessage.aTxData[4])); //Anzahl der zu löschenden Bytes
			fbSendCanMessage.tTimeout := T#3000MS;
			fbSendCanMessage.nTxLength := 8;
			nStateActionNext := 6;
			nStateActionTimeout := 99;
			nStateAction := 60;
			//Erwartete Antwort
			HEXSTR_TO_DATA('FF00000000000000',ADR(aExpectedData),8);
	
		6:	//PROGRAM
			//Blockaufbau
			//F6 XX XX XX XX XX XX XX	(SET_MTA)
			//DO XX XX XX				(PROGRAM)
			//C9 XX XX XX XX XX XX XX	(PROGRAM_MAX)
			//C9 XX XX XX XX XX XX XX	(PROGRAM_MAX)
			//usw
			//Die Blöcke werden von "fbS19File" gebildet
			stInfo.eActState := E_FirmwUpdState.Programming;
			fbS19File.A_FitProgLine(bExecute:= TRUE);
			IF NOT fbS19File.bBusy THEN
				stInfo.nWrittenBytes := fbS19File.P_nWrittenBytes;
				fbSendCanMessage.nTxLength := fbS19File.M_GetProgLine(ADR(fbSendCanMessage.aTxData));
				fbSendCanMessage.tTimeout := T#100MS;
				nStateActionTimeout := 99;
				nStateAction := 60;
				//Erwartete Antwort
				HEXSTR_TO_DATA('FF00000000000000',ADR(aExpectedData),8);
				IF fbS19File.P_bProgLineDone THEN
					fbS19File.A_FitProgLine(bExecute:= FALSE);
					nStateActionNext := 7;		
				END_IF
			END_IF
			
		7:	//PROGRAM (D0 mit SizeParamter 0)
			fbSendCanMessage.aTxData[0] := 16#D0;	//XCP-Command: PROGRAM
			fbSendCanMessage.aTxData[1] := 0;		//Size-Paramter 0
			fbSendCanMessage.tTimeout := T#100MS;
			fbSendCanMessage.nTxLength := 2;
			nStateActionNext := 8;
			nStateActionTimeout := 99;
			nStateAction := 60;
			//Erwartete Antwort
			HEXSTR_TO_DATA('FF00000000000000',ADR(aExpectedData),8);
		
		8:	//PROGRAM_RESET
			fbSendCanMessage.aTxData[0] := 16#CF;	//XCP-Command: PROGRAM_RESET
			fbSendCanMessage.tTimeout := T#10MS;
			fbSendCanMessage.nTxLength := 1;
			//Durch Reset kommt keine Anwort zurück
			IF pFbCanNode > 0 THEN
				nStateActionNext := 9;
				nStateActionTimeout := 9;
			ELSE
				nStateActionNext := 80;
				nStateActionTimeout := 80;
			END_IF
			nStateAction := 60;
			
		9:	//Close File
			fbS19File.A_CloseFile(bExecute:= TRUE);
			IF NOT fbS19File.bBusy THEN
				fbS19File.A_CloseFile(bExecute:= FALSE);
				stInfo.eActState := E_FirmwUpdState.WaitForBootup;
				nStateAction := 10;
			END_IF
			
		10:	//Warten, dass sich Node meldet
			//Timeout einbauen!!!!!!!!!!!!
			
			IF pFbCanNode^.P_nNodeState = 0 THEN
				stInfo.eActState := E_FirmwUpdState.Ready;	
				pFbCanNode^.P_bStopMonitor := FALSE;	//Überwachung des Node aktivieren
				bBusy := FALSE;
				nStateAction := 80;
			END_IF
	END_CASE
	
	IF nStateAction = 60 THEN	//CAN-Message senden
		fbSendCanMessage(nIdentifierTX:= 16#667, nIdentifierRX:= 16#7E1, bExecute:= TRUE);
		IF NOT fbSendCanMessage.bBusy THEN
			IF NOT fbSendCanMessage.bError THEN
				//Response auswerten
				IF fbSendCanMessage.aRxData[0] = 16#FF THEN	//kein Fehler
					IF MEMCMP(ADR(fbSendCanMessage.aRxData),ADR(aExpectedData),8) = 0 THEN
						nStateAction := nStateActionNext;
					ELSE
						nStateAction := 99;
					END_IF
				ELSIF fbSendCanMessage.aRxData[0] = 16#FE THEN	//Error in respone
					CASE fbSendCanMessage.aRxData[1] OF
						16#00:	nErrorId := E_ErrorIdCan.ERRORID_XcpErrCmdSynch;
						16#10:	nErrorId := E_ErrorIdCan.ERRORID_XcpErrCmdBusy;
						16#20:	nErrorId := E_ErrorIdCan.ERRORID_XcpErrCmdUnknown;
						16#22:	nErrorId := E_ErrorIdCan.ERRORID_XcpErrOutOfRange;
						16#25:	nErrorId := E_ErrorIdCan.ERRORID_XcpErrAccessLocked;
						16#26:	nErrorId := E_ErrorIdCan.ERRORID_XcpErrPageNotValid;
						16#29:	nErrorId := E_ErrorIdCan.ERRORID_XcpErrSequence;
						16#31:	nErrorId := E_ErrorIdCan.ERRORID_XcpErrGeneric;
					END_CASE
					nStateAction := 99;
				END_IF
			ELSE
				nStateAction := nStateActionTimeout;
			END_IF
			fbSendCanMessage(bExecute:= FALSE);
		END_IF		
	END_IF
	
	IF nStateAction = 99 THEN
		stInfo.eActState := E_FirmwUpdState.Error;
		//CloseFile
		fbS19File.A_CloseFile(bExecute:= TRUE);
		IF NOT fbS19File.bBusy THEN
			bError := TRUE;
			bBusy := FALSE;
			nStateAction := 100;
		END_IF
	END_IF
ELSE
	nStateAction := 0;
	bError := FALSE;
END_IF

END_PROGRAM

// ---- Hardware/FB_CanNodeBase.TcPOU
FUNCTION_BLOCK FB_CanNodeBase EXTENDS FB_HwModule
VAR_INPUT
END_VAR
VAR_OUTPUT
END_VAR
VAR
	stAdsAdress		: ST_AdsAdress;
	bNodeEnabled	: BOOL;
	bNodeFound		: BOOL;
	nNodeId			: USINT;
	nNodeState		AT %I* : USINT;	//PDO
	nErrorId 		: ERRORID;
	nErrorId2 		: UDINT;
	sHardwVersion	: STRING(15);
	sSoftwVersion	: STRING(15);
	
	bPrepare			: BOOL;
	nStateA_Prepare 	: USINT;
	bPreparingOK		: BOOL;
	
	bResetError		: BOOL;
	nStateResetError: USINT;
	
	bResetApp		: BOOL;
	nStateA_ResetApp: USINT;
	
	fbSdoRead 		: FB_SDO_READ;
	fbSdoWrite		: FB_SDO_WRITE;
	nPOUState 		: USINT;
	
	bStopMonitor	: BOOL;
	
	timeout			: TON;
END_VAR

IF bPrepare THEN
	A_Prepare();
	IF nStateA_Prepare >= 80 THEN
		IF nStateA_Prepare >= 99 THEN
			bError := TRUE;
		ELSE
			bPreparingOK := TRUE;
		END_IF
		nStateA_Prepare := 0;
		bPrepare := FALSE;
	END_IF
END_IF

IF bResetApp THEN
	A_ResetApp();
	IF nStateA_ResetApp >= 80 THEN
		IF nStateA_ResetApp >= 99 THEN
			bError := TRUE;
		END_IF
		nStateA_ResetApp := 0;
		bResetApp := FALSE;
	END_IF
END_IF

bBusy := bPrepare OR bResetError OR bResetApp;

ACTION A_Monitor:
IF nNodeState > 0  THEN
	bError := TRUE;
END_IF
END_ACTION

ACTION A_Prepare:
nPOUState := nStateA_Prepare;
CASE nStateA_Prepare OF
	0:	//Checken, ob Node "operational"
		//Timeout von 10s
		timeout(IN:= TRUE, PT:= T#10S);
		IF nNodeState = 0 THEN
			timeout(IN:= FALSE);
			bNodeFound := TRUE;
			nStateA_Prepare := 1;
		END_IF
		IF timeout.Q THEN
			timeout(IN:= FALSE);
			nStateA_Prepare := 99;
			CASE nNodeState OF
				1:	nErrorId := E_ErrorIdCan.ERRORID_NodeDeactivated;
				2:	nErrorId := E_ErrorIdCan.ERRORID_NodeNotFound;
					//Nur in Fehler gehen, wenn Node die Kopfbasisplatine ist.
					//Ein Error zu folge hätte, dann würde es auch bei einem abgestecktem Mtp-Heater zu einem Error kommen.
					IF stHardwareId.eGroup <> E_HardwareGrp.MultiZBasis THEN
						nStateA_Prepare := 80;	
					END_IF
				4:	nErrorId := E_ErrorIdCan.ERRORID_SdoSyntaxErrorAtStartup;
				5:	nErrorId := E_ErrorIdCan.ERRORID_SdoDataMismatchAtStartup;
				12:	nErrorId := E_ErrorIdCan.ERRORID_NodePreOP;
			END_CASE
		END_IF

	1:	//Hardwareversion auslesen
		fbSdoRead(sADSNetID:= stAdsAdress.sNetId, nPortNr:= stAdsAdress.nPort,
				nIndex:= 16#1009, nSubIndex:= 0, nDataLength:= 20, bExecute:= TRUE);
				
		IF NOT fbSdoRead.bBusy THEN
			IF fbSdoRead.bError THEN
				nErrorId := fbSdoRead.nAdsErrorId;
				nErrorId2 := fbSdoRead.nSdoErrorId;
				nStateA_Prepare := 99;	//Error
			ELSE
				sHardwVersion := fbSdoRead.sData;
				nStateA_Prepare := 2;
			END_IF
			fbSdoRead(bExecute:= FALSE);
		END_IF
		
	2:	//Softwareversion auslesen
		fbSdoRead(sADSNetID:= stAdsAdress.sNetId, nPortNr:= stAdsAdress.nPort,
				nIndex:= 16#100A, nSubIndex:= 0, nDataLength:= 20, bExecute:= TRUE);
				
		IF NOT fbSdoRead.bBusy THEN
			IF fbSdoRead.bError THEN
				nErrorId := fbSdoRead.nAdsErrorId;
				nErrorId2 := fbSdoRead.nSdoErrorId;
				nStateA_Prepare := 99;	//Error
			ELSE
				sSoftwVersion := fbSdoRead.sData;
				nStateA_Prepare := 80;
			END_IF
			fbSdoRead(bExecute:= FALSE);
		END_IF
	
END_CASE

IF nStateA_Prepare = 99 THEN
	stError.Cmd := 0;
	stError.ErrorId := nErrorId;
	stError.HardwareGrp := stHardwareId.eGroup;
	stError.HardwareNr := stHardwareId.nItem;
END_IF
END_ACTION

ACTION A_ResetApp:
nStateA_ResetApp := 80;
END_ACTION

METHOD M_GetHwInfo : ST_HardwareInfo
VAR_INPUT
END_VAR
M_GetHwInfo := SUPER^.M_GetHwInfo();
M_GetHwInfo.sHardwVersion := sHardwVersion;
M_GetHwInfo.sSoftwVersion := sSoftwVersion;
END_METHOD

METHOD M_Prepare
VAR_INPUT
	sAdsNetId	: STRING(23);
	nCanNodeId	: USINT;
END_VAR
stAdsAdress.sNetId := sAdsNetId;
stAdsAdress.nPort := nCanNodeId + 4096;
nNodeId := nCanNodeId;
bNodeEnabled := TRUE;
bPrepare := TRUE;
bPreparingOK := FALSE;
END_METHOD

METHOD M_Reset
VAR_INPUT
END_VAR
IF bError THEN
	bResetError := TRUE;
END_IF
END_METHOD

METHOD M_ResetApp
VAR_INPUT
END_VAR
bResetApp := TRUE;
END_METHOD

PROPERTY P_bNodeEnabled : BOOL
GET
P_bNodeEnabled := bNodeEnabled;
END_GET
END_PROPERTY

PROPERTY P_bStopMonitor : BOOL
GET
P_bStopMonitor := bStopMonitor;
END_GET
SET
bStopMonitor := P_bStopMonitor;
END_SET
END_PROPERTY

PROPERTY P_nAdsPort : UINT
GET
P_nAdsPort := stAdsAdress.nPort;
END_GET
END_PROPERTY

PROPERTY P_nNodeId : USINT
GET
P_nNodeId := nNodeId;
END_GET
END_PROPERTY

PROPERTY P_nNodeState : USINT
GET
P_nNodeState := nNodeState;
END_GET
END_PROPERTY

PROPERTY P_sAdsNetId : STRING(23)
GET
P_sAdsNetId := stAdsAdress.sNetId;
END_GET
END_PROPERTY

PROPERTY P_sHardwVersion : STRING(15)
GET
P_sHardwVersion := sHardwVersion;
END_GET
END_PROPERTY

PROPERTY P_sSoftwVersion : STRING(15)
GET
P_sSoftwVersion := sSoftwVersion;
END_GET
END_PROPERTY

END_FUNCTION_BLOCK

// ---- Hardware/FB_HwModule.TcPOU
FUNCTION_BLOCK FB_HwModule
VAR_INPUT
END_VAR
VAR_OUTPUT
END_VAR
VAR
	stHardwareId : ST_HardwareId;
	bBusy : BOOL;
	bError : BOOL;
	stError : ST_Error;
END_VAR

METHOD M_GetHwInfo : ST_HardwareInfo
VAR_INPUT
END_VAR

VAR
	nHwId : UDINT;
END_VAR
nHwId := SHL(UINT_TO_UDINT(stHardwareId.eGroup),16);
nHwId := nHwId OR (SHL(UINT_TO_UDINT(stHardwareId.nParentItem),8));
nHwId := nHwId OR stHardwareId.nItem;
M_GetHwInfo.nHwId := nHwId;
END_METHOD

METHOD M_Reset
VAR_INPUT
END_VAR
END_METHOD

PROPERTY P_bBusy : BOOL
GET
P_bBusy := bBusy;
END_GET
END_PROPERTY

PROPERTY P_bError : BOOL
GET
P_bError := bError;
END_GET
END_PROPERTY

PROPERTY P_eHardwareGrp : E_HardwareGrp
GET
P_eHardwareGrp := stHardwareId.eGroup;
END_GET
END_PROPERTY

PROPERTY P_stError : ST_Error
GET
P_stError := stError;
END_GET
END_PROPERTY

PROPERTY P_stHardwareId : ST_HardwareId
GET
P_stHardwareId := stHardwareId;
END_GET
SET
stHardwareId := P_stHardwareId;
END_SET
END_PROPERTY

END_FUNCTION_BLOCK

// ---- Hardware/SDO_Com/FB_SDO_READ.TcPOU
FUNCTION_BLOCK FB_SDO_READ
VAR_INPUT
	sADSNetID		: STRING(23); 	//AMSNetID von Klemme EL6751. Can be empty if only one local single channel card is present
    nPortNr			: WORD;         //Port No. vom CANopen-Knoten (siehe Gerätemanager)
    nIndex			: DWORD;      	//ObjectIndex vom zu lesenden CANopen-Objecteintrag
    nSubIndex		: DWORD;   		//SubIndex vom zu lesenden CANopen-Objecteintrag
    nDataLength		: DWORD;   		//Länge des zu lesenden Datums (max 4 Byte)
    bExecute		: BOOL;
END_VAR

VAR_OUTPUT
	bBusy			: BOOL;
	nData			: DINT;
	sData			: STRING(20);
    bError			: BOOL;
    nAdsErrorId		: ERRORID;	//Ads-ErrorId
	nSdoErrorId		: UDINT;	//Sdo-ErrorId
END_VAR

VAR
    nState			: USINT;
    ADSREAD			: ADSREAD;
	uSdoData		: U_SDO_DATA;	//Union mit empfangenen Bytes und entsprechendem DINT
	nCount			: USINT;
END_VAR

IF bExecute THEN
	nCount := nCount + 1;
	
	CASE nState OF
		0:	
			bBusy := TRUE;
			MEMSET(ADR(uSdoData),0,SIZEOF(uSdoData));
			ADSREAD(NETID:= sADSNetID, PORT:= nPortNr, IDXGRP:= nIndex, IDXOFFS:= nSubIndex, 
					LEN:= nDataLength, DESTADDR:= ADR(uSdoData), READ:= TRUE, TMOUT:= T#5S);

			IF ADSREAD.ERR THEN
				bError := TRUE;
				//ADSREAD.ERRID in Ads-Error und Sdo-Error aufsplitten
				// Ads-Error steht in Bit 0-15
				nAdsErrorId := UDINT_TO_UINT(ADSREAD.ERRID AND 16#0000FFFF);
				//Sdo-Error steht in Bit 16-31
				nSdoErrorId := F_AdsError_TO_SdoError(ADSREAD.ERRID);
				//Gelesenes Datum aus Union in Output-Datum übertragen
				nData := uSdoData.nData;
				ADSREAD(READ:= FALSE);
				bBusy := FALSE;
				nState := 99;
			ELSE
				nState := 1;
			END_IF
		1:
			ADSREAD(READ:= FALSE); //Wenn hier schon auf False gesetzt wird, braucht es weniger Zyklen zum lesen

			IF ADSREAD.ERR THEN
				bError := TRUE;
				//ADSREAD.ERRID in Ads-Error und Sdo-Error aufsplitten
				// Ads-Error steht in Bit 0-15
				nAdsErrorId := UDINT_TO_UINT(ADSREAD.ERRID AND 16#0000FFFF);
				//Sdo-Error steht in Bit 16-31
				nSdoErrorId := F_AdsError_TO_SdoError(ADSREAD.ERRID);
				//Gelesenes Datum aus Union in Output-Datum übertragen
				nData := uSdoData.nData;
				sData := uSdoData.sData;
				ADSREAD(READ:= FALSE);
				bBusy := FALSE;
				nState := 99;
			ELSE
				IF NOT ADSREAD.BUSY THEN
					//Gelesenes Datum aus Union in Output-Datum übertragen
					nData := uSdoData.nData;
					sData := uSdoData.sData;
					ADSREAD(READ:= FALSE);
					nState := 2;
					bBusy := FALSE;
				END_IF; 				
			END_IF
	END_CASE
ELSE
	bBusy := FALSE;
	bError := FALSE;
	nAdsErrorId := 0;
	nSdoErrorId := 0;
	nState := 0;
	nData := 0;
	sData := '';
END_IF

END_FUNCTION_BLOCK

// ---- Hardware/SDO_Com/F_AdsError_TO_SdoError.TcPOU
FUNCTION F_AdsError_TO_SdoError : UDINT
VAR_INPUT
	nAdsErrorId		: UDINT;
END_VAR
VAR
	nSdoErrorIdTemp	: UDINT;
END_VAR

//SDO abort-Codes stehen in Bit 16-30
//SDO Additional Code (0..6) in Bit 24-30
nSdoErrorIdTemp := nAdsErrorId AND 16#7F000000;	//maskieren
nSdoErrorIdTemp := SHR(nSdoErrorIdTemp,24);	//24 bit nach rechts verschieben
F_AdsError_TO_SdoError := F_AdsError_TO_SdoError OR nSdoErrorIdTemp;
//SDO Error Code (16..19) in Bit 20-23
nSdoErrorIdTemp := nAdsErrorId AND 16#00F00000;	//maskieren
nSdoErrorIdTemp := SHR(nSdoErrorIdTemp,4);	//4 bit nach rechts verschieben
F_AdsError_TO_SdoError := F_AdsError_TO_SdoError OR nSdoErrorIdTemp;
//SDO Error Class (24..27) in Bit 16-19
nSdoErrorIdTemp := nAdsErrorId AND 16#000F0000;	//maskieren
nSdoErrorIdTemp := SHL(nSdoErrorIdTemp,8);	//8 bit nach links verschieben
F_AdsError_TO_SdoError := F_AdsError_TO_SdoError OR nSdoErrorIdTemp;

END_FUNCTION

// ---- Hardware/SDO_Com/FB_SDO_WRITE.TcPOU
FUNCTION_BLOCK FB_SDO_WRITE
VAR_INPUT
	sADSNetID		: STRING(23); 	//AMSNetID von Klemme EL6751. Can be empty if only one local single channel card is present
	nPortNr			: WORD;         //Port No. vom CANopen-Knoten (siehe Gerätemanager)
	nIndex			: DWORD;      	//ObjectIndex vom zu lesenden CANopen-Objecteintrag
	nSubIndex		: DWORD;   		//SubIndex vom zu lesenden CANopen-Objecteintrag
	nDataLength		: DWORD;   		//Länge des zu lesenden Datums (max 4 Byte)
	nData			: DINT;
	bExecute		: BOOL;
END_VAR

VAR_OUTPUT
	bBusy			: BOOL;
    bError			: BOOL;
    nAdsErrorId		: ERRORID;	//Ads-ErrorId
	nSdoErrorId		: UDINT;	//Sdo-ErrorId	
END_VAR

VAR
	nState			: USINT;
	ADSWRITE		: Tc2_System.ADSWRITE;
	uSdoData		: U_SDO_DATA;	//Union mit zusendenden Bytes und entsprechendem DINT
	nCount			: USINT;
END_VAR

IF bExecute THEN
	nCount := nCount + 1;
	IF nState = 0 THEN
		bBusy := TRUE;
		uSdoData.nData := nData;
		ADSWRITE(NETID:= sADSNetID, PORT:= nPortNr, IDXGRP:= nIndex, IDXOFFS:= nSubIndex, 
				LEN:= nDataLength, SRCADDR:= ADR(uSdoData), WRITE:= TRUE, TMOUT:= T#1S);	
	ELSIF nState = 1 THEN
			ADSWRITE(WRITE:= FALSE); //Wenn hier schon auf False gesetzt wird, braucht es weniger Zyklen zum lesen
	END_IF
	
	IF ADSWRITE.ERR THEN
		//ADSREAD.ERRID in Ads-Error und Sdo-Error aufsplitten
		// Ads-Error steht in Bit 0-15
		nAdsErrorId := UDINT_TO_UINT(ADSWRITE.ERRID AND 16#0000FFFF);
		//Sdo-Error steht in Bit 16-31
		nSdoErrorId := F_AdsError_TO_SdoError(ADSWRITE.ERRID);
		
		//Fals Error = 1802 (out of memory) Schreibvorgang wiederholen
		IF nAdsErrorId = 1802 THEN
			nState := 0;
		ELSE
			bError := TRUE;
			bBusy := FALSE;
			nState := 99;					
		END_IF
		ADSWRITE(WRITE:= FALSE);
	ELSE
		IF NOT ADSWRITE.BUSY THEN
			//Gelesenes Datum aus Union in Output-Datum übertragen
			nData := uSdoData.nData;
			ADSWRITE(WRITE:= FALSE);
			nState := 2;
			bBusy := FALSE;
		END_IF; 				
	END_IF		
ELSE
	bBusy := FALSE;
	bError := FALSE;
	nAdsErrorId := 0;
	nSdoErrorId := 0;
	nState := 0;	
END_IF

END_FUNCTION_BLOCK

// ---- Hardware/FB_SendCanMessage.TcPOU
FUNCTION_BLOCK FB_SendCanMessage
VAR_INPUT
	nIdentifierTX : UINT;
	nIdentifierRX : UINT;
	tTimeout	: TIME;
	nTxLength : USINT;
	aTxData : ARRAY[0..7] OF USINT;
	bExecute : BOOL;
END_VAR
VAR_OUTPUT
	bBusy : BOOL;
	bError : BOOL;
	nErrorId : ERRORID;
	nRxLength : USINT;
	aRxData : ARRAY[0..7] OF USINT;
END_VAR
VAR
	pBuffer : POINTER TO ST_CANInterfaceBuffer;
	nState 	: USINT;
	pSelf 	: PVOID;
	fbList		: FB_LinkedListCtrl;
	tmrTimeout	: TON;
END_VAR

//Dieser Baustein regelt die Kommunikation mit dem CANInterface
//Wenn es mehrere Instanzen gibt, dann muss eigentlich CANInterfaceCom das Dispachen übernehmen
//In der Regel muss auf jede Tx ein Rx erfolgen
IF bExecute THEN
	//am CANInterface anmelden und warten, bis angemeldet
	//Wie am Interface anmelden? In den Buffer die eigene Adresse schreiben
	//dann nachschauen, ob eigende Adresse übernommen wurde, dass ist das Zeichen, dass die Daten von diesem Baustein verarbeitet werden
	//es auf done gewartet
	IF nState = 0 THEN
		//Request an CANInterface
		fbList.A_AddHeadValue(hList:= pBuffer^.hList, putValue:= pSelf);
		nState := 1;
		bBusy := TRUE;
	END_IF
	
	IF nState = 1 THEN	//Checken, ob an der Reihe
		fbList.A_GetTail(hList:= pBuffer^.hList);
		IF fbList.bOk THEN
			IF fbList.getValue = pSelf THEN
				nState := 2;	
			END_IF
		END_IF
	END_IF
	
	IF nState = 2 THEN	//Buffer füllen; Ab hier wird das CANInterface für andere Instanzen dieses Bausteins blockiert
		IF NOT pBuffer^.bExecute THEN
			pBuffer^.nTxIdent := nIdentifierTX;
			pBuffer^.nTxDlc := nTxLength;
			pBuffer^.aTxData := aTxData;
			pBuffer^.bExecute := TRUE;
			nState := 3;
			//Timer starten !!!
			tmrTimeout(IN:= TRUE, PT:= tTimeout);
		END_IF
	ELSIF nState = 3 THEN	//warten bis gesendet und erwarteter RxIdent empfangen
		tmrTimeout();
		IF tmrTimeout.Q THEN
			bError := TRUE;
			nErrorId := E_ErrorIdCan.ERRORID_TimeoutSendCanMsg;
			bBusy := FALSE;
			nState := 99;
			fbList.A_RemoveTailValue(hList:= pBuffer^.hList);
			pBuffer^.bExecute := FALSE;
			RETURN;
		END_IF
		
		IF NOT pBuffer^.bBusy THEN
			IF pBuffer^.bError THEN
				bError := TRUE;
			ELSE //Daten auswerten
				//wenn erwarteter RxIdent nicht übereinstimmt, dann Error
				IF nIdentifierRX = pBuffer^.nRxIdent THEN
					nRxLength := pBuffer^.nRxDlc;
					aRxData := pBuffer^.aRxData;
				ELSE //Error
					bError := TRUE;
					nState := 99;
				END_IF
			END_IF
			fbList.A_RemoveTailValue(hList:= pBuffer^.hList);
			pBuffer^.bExecute := FALSE;
			bBusy := FALSE;
		END_IF
	END_IF
ELSE
	bBusy := FALSE;
	bError := FALSE;
	nState := 0;
	nRxLength := 0;
	MEMSET(ADR(aRxData),0,SIZEOF(aRxData));
	tmrTimeout(IN:= FALSE);
END_IF

METHOD FB_init : BOOL
VAR_INPUT
	bInitRetains : BOOL; // if TRUE, the retain variables are initialized (warm start / cold start)
	bInCopyCode : BOOL;  // if TRUE, the instance afterwards gets moved into the copy code (online change)
	pCANInterfaceBuffer : POINTER TO ST_CANInterfaceBuffer;
END_VAR
THIS^.pBuffer := pCANInterfaceBuffer;
pSelf := THIS;
END_METHOD

END_FUNCTION_BLOCK

// ---- FirmwUpdate/FB_S19File.TcPOU
FUNCTION_BLOCK FB_S19File
VAR_INPUT
	sFileName	: STRING;
	bExecute	: BOOL;
END_VAR
VAR_OUTPUT
	bBusy : BOOL;
	bError : BOOL;
	nErrorId : ERRORID;
END_VAR
VAR
	fbFileOpen	: FB_FileOpen;
	fbFileClose : FB_FileClose;
	fbFileRead  : FB_FileRead;
	fbFileSeek	: FB_FileSeek;
	nFileHandle	: UINT;
	
	
	bStart : R_TRIG;
	nStateA_OpenFile	: USINT;
	nStateA_CloseFile	: USINT;
	
	bIsOpen	: BOOL;

	aBuffer		: ARRAY[1..4700] OF BYTE;
	nRecord		: UINT;
	fbS19Record	: FB_S19Record;
	
	dwAddress			: DWORD;
	dwStartAddress 		: DWORD;
	dwLastAddress 		: DWORD;
	nNoOfTotalBytes 	: UDINT;
	nFirstBlockSize 	: UDINT;
	n256Blocks 			: UDINT;
	nFirstDataLength 	: USINT;
	i 					: USINT;
	
	nActIndex			: UINT;	
	
	
	//Action: A_FitProgLine
	nStateA_FitProgLine	: USINT;
	nStateA_FitProgLine1: USINT;
	aData 				: ARRAY[0..7] OF USINT;
	nBytesToSend 		: USINT;
	
	nWriteBytesLine		: USINT;
	nWriteBytesBlock	: UINT;
	nWriteBytesTotal	: UDINT;
	bProgLineDone		: BOOL;

END_VAR

PROPERTY P_nBytesToWrite : UDINT
GET
P_nBytesToWrite := nNoOfTotalBytes;
END_GET
END_PROPERTY

ACTION A_CloseFile:
IF bExecute THEN
	IF nFileHandle = 0 THEN
		RETURN;
	END_IF
	bBusy := TRUE;
	fbFileClose(hFile:= nFileHandle, bExecute:= TRUE);
	IF NOT fbFileClose.bBusy THEN
		fbFileClose(bExecute:= FALSE);
		bIsOpen := FALSE;
		bBusy := FALSE;
	END_IF
END_IF
END_ACTION

METHOD M_GetProgLine : USINT //Bytes
VAR_INPUT
	pData	: POINTER TO ARRAY[0..7] OF USINT;
END_VAR
MEMCPY(pData,ADR(aData),8);
M_GetProgLine := nBytesToSend;
END_METHOD

METHOD M_GetStartAdress
VAR_INPUT
	pData	: POINTER TO ARRAY[0..7] OF USINT;
END_VAR
MEMCPY(pData,ADR(dwStartAddress),4);
END_METHOD

PROPERTY P_nWrittenBytes : UDINT
GET
P_nWrittenBytes := nWriteBytesTotal;
END_GET
END_PROPERTY

METHOD M_GetNoOfTotalBytes
VAR_INPUT
	pData	: POINTER TO ARRAY[0..7] OF USINT;
END_VAR
IF pData > 0 THEN
	MEMCPY(pData,ADR(nNoOfTotalBytes),4);
END_IF
END_METHOD

PROPERTY P_bProgLineDone : BOOL
GET
P_bProgLineDone := nStateA_FitProgLine1 = 80;
END_GET
END_PROPERTY

ACTION A_OpenFile:
IF bExecute THEN
	CASE nStateA_OpenFile OF
		0:	//Open File
			IF bIsOpen THEN
				bError := TRUE;
				nErrorId := E_ErrorIdCan.ERRORID_FileAlreadyOpened;
				RETURN;
			END_IF
			bBusy := TRUE;
			fbFileOpen(sPathName:= sFileName, nMode:= FOPEN_MODEREAD OR FOPEN_MODETEXT, bExecute:= TRUE, tTimeout:= T#10S);
			IF NOT fbFileOpen.bBusy THEN
				IF fbFileOpen.bError THEN
					nStateA_OpenFile := 99;
					nErrorId := UDINT_TO_UINT(fbFileOpen.nErrId);
				ELSE
					nStateA_OpenFile := 1;
					nFileHandle := fbFileOpen.hFile;
					nRecord := 0;
				END_IF
				fbFileOpen(bExecute:= FALSE);
			END_IF
			
		1:	//Blockweise 100 Zeilen einlesen
			fbFileRead(hFile:= nFileHandle,	pReadBuff:= ADR(aBuffer), cbReadLen:= SIZEOF(aBuffer), bExecute:= TRUE);
			IF NOT fbFileRead.bBusy THEN
				IF fbFileRead.bError THEN
					nStateA_OpenFile := 99;
				ELSE
					nActIndex := 0;
					REPEAT
						nActIndex := nActIndex + 1;
						fbS19Record(pBuffer:= ADR(aBuffer), nStartIndex:= nActIndex, nEndIndex=> nActIndex);
						CASE fbS19Record.eState OF
							E_S19RecordState.Valid:
								nRecord := nRecord + 1;
								IF nRecord = 1 THEN
									dwStartAddress := fbS19Record.P_dwAdress;
								END_IF
								dwLastAddress := fbS19Record.P_dwAdress;
							E_S19RecordState.BlockEnd:
								nNoOfTotalBytes := (dwLastAddress - dwStartAddress + fbS19Record.P_nNoOfDataBytes);
								nFirstBlockSize := nNoOfTotalBytes MOD 256;
								n256Blocks := (nNoOfTotalBytes - nFirstBlockSize) / 256;
								nFirstDataLength := UDINT_TO_USINT(nFirstBlockSize MOD 7);
								nStateA_OpenFile := 2;
								EXIT;
							E_S19RecordState.NotComplete:
								//dürfte eingentlich nicht eintreten
								nErrorId := E_ErrorIdCan.ERRORID_FirmwFileCorrupt;
								nStateA_OpenFile := 99;
								EXIT;
							E_S19RecordState.CRC_Error:
								nErrorId := E_ErrorIdCan.ERRORID_FirmwFileCRCError;
								nStateA_OpenFile := 99;
								EXIT;
							E_S19RecordState.Line_Error:
								nErrorId := E_ErrorIdCan.ERRORID_FirmwFileLineError;
								nStateA_OpenFile := 99;
								EXIT;
							E_S19RecordState.Undefined:
								nStateA_OpenFile := 99;
								EXIT;
						END_CASE
					UNTIL fbS19Record.bEndOfBuffer
					END_REPEAT
				END_IF
				IF fbFileRead.bEOF THEN
					nErrorId := E_ErrorIdCan.ERRORID_FirmwFileEOF;
					nStateA_OpenFile := 99;
				END_IF
				MEMSET(ADR(aBuffer),0,SIZEOF(aBuffer));
				fbFileRead(bExecute:= FALSE);
			END_IF
		
		2:	//Datei-Zeiger wieder auf "0" stellen
			fbFileSeek(hFile:= nFileHandle,	nSeekPos:= 0, bExecute:= TRUE);
			IF NOT fbFileSeek.bBusy THEN
				fbFileSeek(bExecute:= FALSE);
				bIsOpen := TRUE;
				nStateA_OpenFile := 80;
				bBusy := FALSE;
			END_IF
	END_CASE
	
	IF nStateA_OpenFile = 99 THEN
		bError := TRUE;
		bBusy := FALSE;
		fbFileClose(hFile:= nFileHandle, bExecute:= TRUE);
		fbFileClose(hFile:= nFileHandle, bExecute:= FALSE);	
	END_IF
	
ELSE
	bError := FALSE;
	nErrorId := 0;
	nStateA_OpenFile := 0;
END_IF
END_ACTION

ACTION A_FitProgLine:
bStart(CLK:= bExecute);
IF bStart.Q AND nStateA_FitProgLine = 0 THEN
	nStateA_FitProgLine := 1;
	nStateA_FitProgLine1 := 0;
	fbS19Record.M_Clear();
	nWriteBytesLine	 := 1;
	nWriteBytesBlock := 0;
	nWriteBytesTotal := 0;
END_IF

IF nStateA_FitProgLine = 1 THEN	//nächsten Block in den Buffer laden
	bBusy := TRUE;
	fbFileRead(hFile:= nFileHandle,	pReadBuff:= ADR(aBuffer), cbReadLen:= SIZEOF(aBuffer), bExecute:= TRUE);
	IF NOT fbFileRead.bBusy THEN
		IF fbFileRead.bError THEN
			nStateA_FitProgLine := 99;
		ELSE
			nStateA_FitProgLine := 2;
		END_IF
		fbFileRead(bExecute:= FALSE);
		nActIndex := 0;
	END_IF
END_IF

IF nStateA_FitProgLine = 2 THEN	//nächste Programmzeile zusammensetzen
	IF fbS19Record.P_dwAdress = 0 THEN	//Record füllen
		IF fbS19Record.bEndOfBuffer THEN
			fbS19Record.M_Clear();
			nStateA_FitProgLine := 1;	//nächsten Block einlesen
			bBusy := TRUE;
			RETURN;
		END_IF		
		nActIndex := nActIndex + 1;
		fbS19Record(pBuffer:= ADR(aBuffer), nStartIndex:= nActIndex, nEndIndex=> nActIndex);
	END_IF
	
	CASE nStateA_FitProgLine1 OF
		0:	//MTA für ersten Block
			MEMSET(ADR(aData),0,7);
			aData[0] := 16#F6;	//XCP-Command: SET_MTA
			MEMCPY(ADR(aData[4]),ADR(dwStartAddress),4);
			nBytesToSend := 8;
			
			bBusy := FALSE;
			nStateA_FitProgLine1 := 1;

		1:	//erste Programmzeile erster Block
			bBusy := FALSE;
			IF nFirstDataLength = 0 THEN	//Voller Datensatz mit 7 Bytes
				aData[0] := 16#C9;
				FOR nWriteBytesLine := nWriteBytesLine TO 7 BY 1 DO
					IF fbS19Record.P_dwAdress > 0 THEN
						aData[nWriteBytesLine] := fbS19Record.M_GetDataByte();
						nWriteBytesBlock := nWriteBytesBlock + 1;
						nWriteBytesTotal := nWriteBytesTotal + 1;
					ELSE
						bBusy := TRUE;
						EXIT;
					END_IF
				END_FOR
				nBytesToSend := 8;
			ELSE
				MEMSET(ADR(aData),0,7);
				aData[0] := 16#D0;
				aData[1] := nFirstDataLength;
				FOR nWriteBytesLine := nWriteBytesLine TO nFirstDataLength BY 1 DO
					IF fbS19Record.P_dwAdress > 0 THEN
						aData[nWriteBytesLine + 1] := fbS19Record.M_GetDataByte();
						nWriteBytesBlock := nWriteBytesBlock + 1;
						nWriteBytesTotal := nWriteBytesTotal + 1;
					ELSE
						bBusy := TRUE;
						EXIT;
					END_IF
				END_FOR
				nBytesToSend := nFirstDataLength + 2;
			END_IF
			
			IF nFirstBlockSize < 7 THEN
				nStateA_FitProgLine1 := 3;
			ELSE
				nStateA_FitProgLine1 := 2;
			END_IF			
			
			(*IF NOT bBusy THEN
				nStateA_FitProgLine1 := 2;
			END_IF*)
		
		2:	//restliche Programmzeilen erster Block
			bBusy := FALSE;
			aData[0] := 16#C9;	//XCP-Command: PROGRAM
			FOR nWriteBytesLine := nWriteBytesLine TO 7 BY 1 DO
				IF fbS19Record.P_dwAdress > 0 THEN
					aData[nWriteBytesLine] := fbS19Record.M_GetDataByte();
					nWriteBytesBlock := nWriteBytesBlock + 1;
					nWriteBytesTotal := nWriteBytesTotal + 1;
				ELSE
					bBusy := TRUE;
					EXIT;
				END_IF
			END_FOR
			nBytesToSend := 8;
			//Wann ist der erste Block voll?
			IF nWriteBytesBlock = nFirstBlockSize THEN
				nStateA_FitProgLine1 := 3;
			ELSIF nWriteBytesTotal = nNoOfTotalBytes THEN
				nStateA_FitProgLine := 80;
			END_IF
		
		3:	//MTA für 256Byte-Blöcke
			MEMSET(ADR(aData),0,7);
			bBusy := TRUE;
			IF fbS19Record.P_dwAdress > 0 THEN
				aData[0] := 16#F6;	//XCP-Command: SET_MTA
				dwAddress := fbS19Record.P_dwAdress;
				MEMCPY(ADR(aData[4]),ADR(dwAddress),4);
				nBytesToSend := 8;
				bBusy := FALSE;
				nWriteBytesBlock := 0;
				nStateA_FitProgLine1 := 4;
			END_IF
			
		4:	//erste Programmzeile 256Byte-Blöcke
			bBusy := FALSE;
			aData[0] := 16#D0;
			aData[1] := 4;  //immer 4 Byte
			aData[6] := 0;
			aData[7] := 0;
			FOR nWriteBytesLine := nWriteBytesLine TO 4 BY 1 DO
				IF fbS19Record.P_dwAdress > 0 THEN
					aData[nWriteBytesLine + 1] := fbS19Record.M_GetDataByte();
					nWriteBytesBlock := nWriteBytesBlock + 1;
					nWriteBytesTotal := nWriteBytesTotal + 1;
				ELSE
					bBusy := TRUE;
					EXIT;
				END_IF
			END_FOR
			nBytesToSend := 6;
			IF NOT bBusy THEN
				nStateA_FitProgLine1 := 5;
			END_IF
			
		5:	//restliche Programmzeilen 256Byte-Blöcke
			dwAddress := fbS19Record.P_dwAdress;
			IF dwAddress >= 16#08004C70 THEN
				dwAddress := dwAddress;
			END_IF
			bBusy := FALSE;
			aData[0] := 16#C9;	//XCP-Command: PROGRAM
			IF nWriteBytesTotal = 195 THEN
				nWriteBytesTotal := nWriteBytesTotal;
			END_IF
			FOR nWriteBytesLine := nWriteBytesLine TO 7 BY 1 DO
				IF fbS19Record.P_dwAdress > 0 THEN
					aData[nWriteBytesLine] := fbS19Record.M_GetDataByte();
					nWriteBytesBlock := nWriteBytesBlock + 1;
					nWriteBytesTotal := nWriteBytesTotal + 1;
				ELSE
					bBusy := TRUE;
					EXIT;
				END_IF
			END_FOR
			nBytesToSend := 8;
			//Wann ist Block voll?
			IF nWriteBytesTotal = nNoOfTotalBytes THEN	//Ready!!
				nStateA_FitProgLine := 0;
				nStateA_FitProgLine1 := 80;
			ELSIF nWriteBytesBlock = 256 THEN
				nWriteBytesBlock := 0;
				nStateA_FitProgLine1 := 3;
			END_IF
	END_CASE
END_IF

IF NOT bBusy THEN
	nWriteBytesLine := 1;
END_IF
END_ACTION

END_FUNCTION_BLOCK

// ---- FirmwUpdate/FB_S19Record.TcPOU
FUNCTION_BLOCK FB_S19Record
VAR_INPUT
	pBuffer : POINTER TO ARRAY[1..4700] OF BYTE;
	nStartIndex : UINT;
END_VAR
VAR_OUTPUT
	nEndIndex 		: UINT;
	bEndOfBuffer	: BOOL;
	eState			: E_S19RecordState;
END_VAR
VAR
	nNoOfBytes	: USINT;
	dwStartAdress : DWORD;
	nDataPointer : USINT;
	aData	: ARRAY[0..21] OF BYTE;
	
	sHex2		: STRING[2];
	sHex8		: STRING[8];
	sCRCData	: STRING[45];
	nCRC 		: BYTE;
	i 			: USINT;
END_VAR

bEndOfBuffer := FALSE;
nEndIndex := 0;
eState := E_S19RecordState.Undefined;
IF pBuffer = 0 THEN
	RETURN;
END_IF
//Datensatz aus Buffer extrahieren
//Folgende Resultate sind möglich
//1.Zeilenumbruch ermittelt
//2.Zeilenumbruch ermittelt und Ende vom Buffer
//3.Ende vom Buffer aber kein Zeilenvorschub 'LF'
nEndIndex := nStartIndex;
REPEAT
	nEndIndex := nEndIndex + 1;
UNTIL (nEndIndex = 4700 OR pBuffer^[nEndIndex] = 10)	//Ende des Buffers oder Zeilenvorschub erreicht (10 = ASCII 'LF')
END_REPEAT

IF nEndIndex = 4700 THEN
	bEndOfBuffer := TRUE;
END_IF

IF pBuffer^[nEndIndex] = 10 THEN //LF - vollständiger Datensatz ermittelt -> verifizieren
	MEMCPY(ADR(sHex2),ADR(pBuffer^[nStartIndex]),2);	//Linetype emitteln
	IF sHex2 = 'S3' THEN
		//Anzahl der Bytes extrahieren (Zeichen 3+4)
		MEMCPY(ADR(sHex2),ADR(pBuffer^[nStartIndex + 2]),2);
		HEXSTR_TO_DATA(sHex2,ADR(nNoOfBytes),1);
		//Checksumme bilden
		MEMCPY(ADR(sCRCData),ADR(pBuffer^[nStartIndex + 2]),44); //Die Checksumme wird ab Zeichen 3 gebildet
		HEXSTR_TO_DATA(sCRCData,ADR(aData),22);
		nCRC := 0;
		FOR i:= 0 TO nNoOfBytes - 1 BY 1 DO
			nCRC := nCRC + aData[i];
		END_FOR
		nCRC := NOT nCRC;
		//Checksumme prüfen
		IF nCRC = aData[nNoOfBytes] THEN
			MEMCPY(ADR(sHex8),ADR(pBuffer^[nStartIndex + 4]),8); //StartAdresse Zeichen 5-12
			HEXSTR_TO_DATA(sHex8,ADR(aData),4);
			dwStartAdress := SHL(BYTE_TO_DWORD(aData[0]),24);
			dwStartAdress := dwStartAdress + SHL(BYTE_TO_DWORD(aData[1]),16);
			dwStartAdress := dwStartAdress + SHL(BYTE_TO_DWORD(aData[2]),8);
			dwStartAdress := dwStartAdress + aData[3];
			nDataPointer := 0;
			eState := E_S19RecordState.Valid;
		ELSE
			eState := E_S19RecordState.CRC_Error;
		END_IF
	ELSIF sHex2 = 'S7' THEN
		eState := E_S19RecordState.BlockEnd;
	ELSE
		eState := E_S19RecordState.Line_Error;
	END_IF
ELSE
	eState := E_S19RecordState.NotComplete;
END_IF

PROPERTY P_nNoOfDataBytes : USINT
GET
//Reine Anzahl der Datanbytes (ohne Adresse usw)
P_nNoOfDataBytes := nNoOfBytes - 5;
END_GET
END_PROPERTY

METHOD M_Clear
VAR_INPUT
END_VAR
bEndOfBuffer := FALSE;
nEndIndex := 0;
eState := E_S19RecordState.Undefined;
nNoOfBytes := 0;
dwStartAdress := 0;
nDataPointer := 0;
END_METHOD

METHOD M_GetDataByte : BYTE
VAR_INPUT
END_VAR
VAR_OUTPUT
END_VAR
VAR
	sHex2	: STRING[2];
	nByte	: BYTE;
END_VAR
//Die Datenbytes beginne ab Zeichen 13
//es können maximal 16 Datenbytes sein
IF pBuffer > 0 THEN
	MEMCPY(ADR(sHex2),ADR(pBuffer^[nStartIndex + 12 + (nDataPointer * 2)]),2);
	HEXSTR_TO_DATA(sHex2,ADR(nByte),1);
	nDataPointer := nDataPointer + 1;
	M_GetDataByte := nByte;
END_IF
END_METHOD

PROPERTY P_dwAdress : DWORD
GET
IF nDataPointer <= (nNoOfBytes - 6) THEN
	P_dwAdress := dwStartAdress + nDataPointer;
END_IF
END_GET
END_PROPERTY

END_FUNCTION_BLOCK

// ---- GCode/GCode.TcPOU
PROGRAM GCode
VAR
	//NCI-Funktionsbausteine	
	fbItpLoadProgEx 			: Tc2_NCI.ItpLoadProgEx;
	fbItpResetEx2				: Tc2_NCI.ItpResetEx2;
	fbItpStartStopEx			: Tc2_NCI.ItpStartStopEx;
	fbItpWriteZeroShiftEx		: Tc2_NCI.ItpWriteZeroShiftEx;
	fbItpSetCyclLrealOffs		: Tc2_NCI.ItpSetCyclicLrealOffsets;
	fbItpSetCyclUdintOffs		: Tc2_NCI.ItpSetCyclicUdintOffsets;
	fbItpEStopEx				: Tc2_NCI.ItpEStopEx;
	fbItpStepOnAfterEStopEx 	: Tc2_NCI.ItpStepOnAfterEStopEx;
	fbItpSingleBlock			: Tc2_NCI.ItpSingleBlock;
	fbItpWriteRParams			: Tc2_NCI.ItpWriteRParamsEx;
	fbItpEnableDefaultGCode		: Tc2_NCI.ItpEnableDefaultGCode;		//für Rotation der auszuführenden NC- Programme
	fbItpBlockSearch			: Tc2_NCI.ItpBlockSearch;				//TODO: rauslöchen, wenn im NC Programm der R Parameter nicht mehr auf "0" gesetzt wird. 
	fbMcPower					: Tc2_MC2.MC_Power;
	fbAdsWrite					: ADSWRITE;
	fbEnumFindFileEntry			: FB_EnumFindFileEntry;
	stFindFile					: ST_FindFileEntry;
	stGCodeRef					: ST_GCodeRef;
	pXDrive						: POINTER TO FB_XYDriveBase;
	pYDrive						: POINTER TO FB_XYDriveBase;
	nCyclCounter				: UINT;
	nCyclThreshold				: UINT := 1000;
	
	//Allgemeine-Variablen
	nState				: USINT;
	sGCodeFile			: STRING;
	stInfo				: ST_GCodeInfo;
	stInfo2				: ST_GCodeInfo2;
	aRParamInit			: ARRAY[0..9] OF LREAL;
	lrAngle				: LREAL;
	
	dwAdsValue			: DWORD;
	nProgress			: UINT;
	stMethResult 		: ST_MethResult;
	pTarget				: POINTER TO FB_TargetBase;	//Startpunkt
	pHighVoltTray		: POINTER TO FB_HighVoltTray;
	pTempTool			: POINTER TO FB_MzTool;
	pMesCartDisp		: POINTER TO FB_CartDispenser;
	pTwinPiezoHolder	: POINTER TO FB_TwinPiezoHolder;
	pGCodeTool			: POINTER TO FB_GCodeTool;
	bWriteZeroShift		: BOOL;
	
	bReadFileOffset		: BOOL;
	fbAdsRead			: ADSREAD;
	bAdsError			: BOOL;
	stFileOffsetData	: ST_NciInfo;		
	nFileOffset			: UDINT;
	
	bMoveActionsLocked	: BOOL;
	
	bStop				: BOOL;
	bNciAvailable 		: BOOL;
	
	sAxesList			: Tc2_Nci.ST_ItpAxes;
	eSingleBlockMode	: Tc2_Nci.E_ItpSingleBlockMode;
	stError 			: ST_Error := (POU := E_POU.POU_GCode);
	
	iter				: FB_ObjCollectIterator;
	iterDeep			: FB_ObjCollectIteratorDeep;

	//*****Action-Variablen*****
	
	//Common
	nStateA_Common 		: USINT;
	nStateA_CommonNext	: USINT;

	//A_BuildGroup + A_ClearGroup
	fbBuildGroup		: FB_BuildGroup;
	fbClearGroup		: FB_ClearGroup;
	
	stActionDataMoveZ	: ST_ActionData;
	stActionData		: ST_ActionData;
	
	fbHskMFunc			: FB_HskMFunc;
	fbFastMFunc			: FB_FastMFunc;
	fbRestartPrintAct	: FB_RestartPrintAction;
	
	//A_Pause
	nStateA_Pause		: USINT;
	stCurrentPos		: ST_3DPoint;
	bLockPause			: BOOL;
	
	nSpeed				: DINT;
	
	//Verkettete Liste für ausführbare Actions im State "Pause"
	fbList				: FB_LinkedListCtrl;
	hList				: T_HLINKEDLIST;
	aNodes  			: ARRAY[0..6] OF T_LinkedListEntry;
	getValue			: UDINT;
	getPosPtr       	: POINTER TO T_LinkedListEntry := 0;
	////////////////////////////////////////////////////////////
	
END_VAR
VAR CONSTANT
	cPathWIN_10			: STRING := 'C:\ftp\GCode\';
	cPathWIN_EMBEDDED	: STRING := 'Hard Disk\ftp\GCode\';
	cMaxGCodeTools		: USINT := 20;
	cMaxGCodeTargets	: USINT := 20;
END_VAR

VAR_OUTPUT
	bBusy			: BOOL;
	bError  		: BOOL;
	eGCodeState		: E_GCodeState;
	bNciModeActive	: BOOL; 
END_VAR

IF bWriteZeroShift THEN //Nullpunktverschiebung während der GCode läuft (durch Action "ShiftGCodeZPos")
	fbItpWriteZeroShiftEx(bExecute:= TRUE, sNciToPlc:= stGCodeRef.sNciToPlc, nZsNo:= 54, sZeroShiftDesc:= stGCodeRef.sZeroShiftDesc);
	IF NOT fbItpWriteZeroShiftEx.bBusy THEN
		fbItpWriteZeroShiftEx(bExecute:= FALSE, sNciToPlc:= stGCodeRef.sNciToPlc, nZsNo:= 54, sZeroShiftDesc:= stGCodeRef.sZeroShiftDesc);
		bWriteZeroShift := FALSE;
	END_IF	
END_IF

CASE nState OF
	0:	//Init
		bBusy := TRUE;
		A_Init();
		IF nStateA_Common >= 80 THEN
			IF nStateA_Common >= 99 THEN
				nState := 99;
			ELSE
				nState := 1;
			END_IF
			nStateA_Common := 0;
			bBusy := FALSE;
		END_IF

	1:	//Idle (Warte-Zustand)
		stInfo.eGCodeState := eGCodeState := E_GCodeState.GCodeState_Idle;
		//Aus diesem Zustand wird duch Methode M_Start(..) in "Loading" geschaltet
		bBusy := FALSE;
		bMoveActionsLocked := FALSE;
	
	2:	//Loading GCode-File
		stInfo.eGCodeState := eGCodeState := E_GCodeState.GCodeState_Loading;
		nFileOffset := 0;
		bBusy := TRUE;
		bMoveActionsLocked := TRUE;
		A_Load();
		IF nStateA_Common >= 80 THEN
			IF nStateA_Common >= 99 THEN
				nState := 99;
			ELSE
				IF bStop THEN
					nState := 1;
				ELSE
					nState := 3;
				END_IF
				
			END_IF
			nStateA_Common := 0;
		END_IF
	
	3:	//Starting
		stInfo.eGCodeState := eGCodeState := E_GCodeState.GCodeState_Starting;
		A_Start();
		IF nStateA_Common >= 80 THEN
			IF nStateA_Common >= 99 THEN
				nState := 99;
			ELSE
				nState := 4;
			END_IF
			nStateA_Common := 0;
		END_IF
	
	4:	//Running (Waiting for HSK-Funktions)
		bReadFileOffset := TRUE;
		stInfo.eGCodeState := eGCodeState := E_GCodeState.GCodeState_Running;
		A_Run();
		IF nStateA_Common >= 80 THEN
			IF nStateA_Common >= 99 THEN
				nState := 99;
			ELSE
				nState := 1;	//zurück in Idle
			END_IF
			nStateA_Common := 0;
		END_IF		
	
	5:	//PauseRequest
		stInfo.eGCodeState := eGCodeState := E_GCodeState.GCodeState_PauseRequest;
		A_Pause();
		IF nStateA_Common >= 80 THEN
			IF nStateA_Common >= 99 THEN
				nState := 99;
			ELSE
				IF stInfo.nNciState = Tc2_NCI.NCI_INTERPRETER_READY THEN
					nState := 1;	//weiter Idle
				ELSE
					nState := 6;	//weiter zu 6	
				END_IF
				
			END_IF
			nStateA_Common := 0;
		END_IF
	
	6:	//Pause
		bMoveActionsLocked := FALSE;
		stInfo.eGCodeState := eGCodeState := E_GCodeState.GCodeState_Pause;
		IF bStop THEN
			IF fbHskMFunc.bBusy THEN
				fbHskMFunc(stGCodeRef:= stGCodeRef,pXDrive:= pXDrive, pYDrive:= pYDrive, bStop:= TRUE);
			END_IF
			fbItpEStopEx(sNciToPlc:= GCode.stGCodeRef.sNciToPlc, bExecute:= TRUE);
			IF NOT fbItpEStopEx.bBusy THEN
				IF fbItpEStopEx.bErr THEN
					stError.ErrorId := UDINT_TO_UINT(fbItpEStopEx.nErrId);
					nState := 99;
				ELSE
					nState := 1;
					fbHskMFunc(stGCodeRef:= stGCodeRef, pXDrive:= pXDrive, pYDrive:= pYDrive, bStop:= FALSE, bPause := FALSE, bContinue:= FALSE);
				END_IF
				fbItpEStopEx(sNciToPlc:= GCode.stGCodeRef.sNciToPlc, bExecute:= FALSE);
				bStop := FALSE;
			END_IF
		END_IF
		
	7:	//Continue
		bReadFileOffset := TRUE;
		stInfo.eGCodeState := eGCodeState := E_GCodeState.GCodeState_ContinueRequest;
		A_Continue();
		IF nStateA_Common >= 80 THEN
			IF nStateA_Common >= 99 THEN
				nState := 99;
			ELSE
				nState := 4;	//weiter zu 4 (Running)
			END_IF
			nStateA_Common := 0;
		END_IF			
	
	60:	//Reset
		bBusy := TRUE;
		A_Reset();
		IF nStateA_Common >= 80 THEN
			IF nStateA_Common >= 99 THEN
				nState := 99;
			ELSE
				nState := 1;
			END_IF
			nStateA_Common := 0;
			bBusy := FALSE;
		END_IF		
	
END_CASE

IF nState = 99 THEN
	stInfo.eGCodeState := eGCodeState := E_GCodeState.GCodeState_Error;
	bBusy := FALSE;
	bError := TRUE;
END_IF

//FileOffset für info auslesen
IF bReadFileOffset THEN
	fbAdsRead(PORT:= 501, IDXGRP:= 16#2100 + ItpGetChannelId(stGCodeRef.sNciToPlc), IDXOFFS:= 16#12, 
					LEN:= SIZEOF(stFileOffsetData), DESTADDR:= ADR(stFileOffsetData), READ:= TRUE);
	IF NOT fbAdsRead.BUSY THEN
		IF fbAdsRead.ERR THEN
			bAdsError := TRUE;
		END_IF
		bReadFileOffset := FALSE;
		fbAdsRead(READ:= FALSE);
		
		IF stFileOffsetData.FileOffset > 0 AND stFileOffsetData.FileOffset <= stFindFile.fileSize.dwLowPart THEN
			nFileOffset := stFileOffsetData.FileOffset;
			nProgress := UDINT_TO_UINT((100 * nFileOffset) / stFindFile.fileSize.dwLowPart);	
		END_IF
	END_IF
END_IF
stInfo.nNciState := ItpGetStateInterpreter(GCode.stGCodeRef.sNciToPlc);

stInfo.nFileOffset := nFileOffset;

IF GCode.stGCodeRef.pCurrentTool > 0 THEN
	stInfo.nCurrentObj := GCode.stGCodeRef.pCurrentTool^.P_nObjectID;
END_IF

ACTION A_Continue:
//HSKMFunc in Pause, dann diese nur fortsetzen
//In diesem Fall wurde der Interpreter nicht gestoppt, da HSKMFunc noch nicht bestätigt wurde
IF fbHskMFunc.bIsInPause THEN
	fbHskMFunc(stGCodeRef:= stGCodeRef, pXDrive:= pXDrive, pYDrive:= pYDrive, bContinue := TRUE, bPause:= FALSE, bStop:= FALSE);
	nStateA_Common := 80;
	RETURN;
ELSE
	fbHskMFunc(stGCodeRef:= stGCodeRef, pXDrive:= pXDrive, pYDrive:= pYDrive, bContinue := FALSE, bPause:= FALSE, bStop:= FALSE);
END_IF

CASE nStateA_Common OF
	0:	//Head freifahren
		//MES-Cartridge vorhanden?, MES-Tray vorhanden?, HV eingeschalten?, steht MES-Cartridge über MES-Tray?
		pMesCartDisp := 0;
		pHighVoltTray := pTarget^.M_GetFirstParentOfType(E_ObjectType.OBJECTTYPE_HighVoltTray); 
		IF pHighVoltTray > 0 THEN
			IF pHighVoltTray^.P_nCurrentVoltage > 0 THEN
				stGCodeRef.pHead^.P_pObjCollectNode^.nodes.M_GetIterator(iter);
				WHILE iter.pNode > 0 DO
					IF iter.pNode^.P_pObject > 0 AND_THEN iter.pNode^.P_pObject^.M_bIsGroup(E_ObjectGroup.OBJECTGROUP_MzTool) THEN
						pTempTool := iter.pNode^.P_pObject;
						IF pTempTool^.P_eObjectType = E_ObjectType.OBJECTTYPE_CartDispenser OR
																pTempTool^.P_eObjectType = E_ObjectType.OBJECTTYPE_CartDispStirrer THEN
							IF pTempTool^.P_bIsMESTool THEN
								IF F_PointInnerRect(pTempTool^.P_stCurrentPosPhys,pHighVoltTray^.P_stAbsRect) THEN
									//Dieses Tool wird vom nachfolgendem Freifahren ausgeschlossen
									pMesCartDisp := pTempTool;
									EXIT;
								END_IF
							END_IF
						END_IF
					END_IF				
					iter.M_Increment();
				END_WHILE
			END_IF
		END_IF
		
		bMoveActionsLocked := TRUE;
		stError.ErrorId := stGCodeRef.pHead^.M_MoveFree(pMesCartDisp);
		
		IF stError.ErrorId > 0 THEN
			nStateA_Common := 99;
		ELSE
			nStateA_Common := 1;
		END_IF

	1:	//Head frei?
		IF NOT stGCodeRef.pHead^.M_GetActionBusy(E_Action.ACTION_MoveZ) THEN
			IF stGCodeRef.pCurrentTool > 0 THEN
				IF stGCodeRef.pCurrentTool^.P_eObjectType = E_ObjectType.OBJECTTYPE_TwinPiezoHolder THEN
					pTwinPiezoHolder := stGCodeRef.pCurrentTool;
					IF pTwinPiezoHolder^.P_eCurrentSwivelState <> E_SwivelState.Swiveled THEN
						nStateA_Common := 2; //weiter zu Einschwenken
					ELSE
						nStateA_Common := 4; //weiter zu letzten Punkt fahren
					END_IF
				ELSIF pMesCartDisp > 0 THEN
					nStateA_Common := 7; //weiter zu Gruppe bilden
				ELSE
					nStateA_Common := 4; //weiter zu letzten Punkt fahren
				END_IF
				
			ELSE
				nStateA_Common := 7; //weiter zu Gruppe bilden
			END_IF
		END_IF

		IF stGCodeRef.pHead^.P_bError THEN
			stError.ErrorId := stGCodeRef.pHead^.P_nErrorId;
			stError.ObjectId := stGCodeRef.pHead^.P_nObjectID;
			nStateA_Common := 99;
		END_IF
		
	2:	//TwinPiezoHolder einschwenken
		MEMSET(ADR(stActionData),0,SIZEOF(stActionData));
		stActionData.eAction := E_Action.ACTION_Swivel;
		stActionData.aParams[1] := 1;
		stError.ErrorId := pTwinPiezoHolder^.M_ExeAction(stActionData);
		IF stError.ErrorId > 0 THEN
			nStateA_Common := 99;
		ELSE
			nStateA_Common := 3;
		END_IF
		
	3:	//TwinPiezoHolder eingeschwenkt?
		IF NOT pTwinPiezoHolder^.M_GetActionBusy(E_Action.ACTION_Swivel) THEN
			IF pTwinPiezoHolder^.P_bError THEN
				stError.ErrorId := pTwinPiezoHolder^.P_nErrorId;
				nStateA_Common := 99;
			ELSE
				nStateA_Common := 4;
			END_IF
		END_IF
		
	4:	//zu letzem Punkt zurückfahren
		IF pMesCartDisp > 0 THEN
			nSpeed := 10000;
		ELSE
			nSpeed := -1;
		END_IF
		stActionData.eAction := E_Action.ACTION_MoveXY;
		stActionData.aParams[1] := E_MoveMode.MODE_AbsWithOffset;
		stActionData.aParams[2] := REAL_TO_DINT(stCurrentPos.X);
		stActionData.aParams[3] := REAL_TO_DINT(stCurrentPos.Y);
		stActionData.aParams[4] := nSpeed;
		stActionData.aParams[5] := nSpeed;
		
		stError.ErrorId := stGCodeRef.pCurrentTool^.M_ExeAction(stActionData);
		IF stError.ErrorId > 0 THEN
			nStateA_Common := 99;
		ELSE
			nStateA_Common := 5;
		END_IF	

	5:	//MoveXY ready? -> MoveZ
		IF NOT stGCodeRef.pCurrentTool^.M_GetActionBusy(E_Action.ACTION_MoveXY) THEN
			MEMSET(ADR(stActionData),0,SIZEOF(stActionData));
			stActionData.eAction := E_Action.ACTION_MoveZ;
			stActionData.aParams[1] := E_MoveMode.MODE_AbsWithOffset;
			stActionData.aParams[2] := REAL_TO_DINT(stCurrentPos.Z);
			stActionData.aParams[3] := nSpeed;
			
			stError.ErrorId := stGCodeRef.pCurrentTool^.M_ExeAction(stActionData);
			IF stError.ErrorId > 0 THEN
				nStateA_Common := 99;
			ELSE
				nStateA_Common := 6;
			END_IF			
		END_IF

	6:	//MoveZ ready?
		IF NOT stGCodeRef.pCurrentTool^.M_GetActionBusy(E_Action.ACTION_MoveZ) THEN
			nStateA_Common := 7;
			IF stGCodeRef.pHead^.P_pXDrive^.P_bIsMoving OR stGCodeRef.pHead^.P_pYDrive^.P_bIsMoving THEN
				nStateA_Common := 6;
			END_IF
		END_IF
		
	7:	//Gruppe bilden
		fbBuildGroup(stGCodeRef:= stGCodeRef, bExecute:= TRUE);
		IF NOT fbBuildGroup.bBusy THEN
			IF fbBuildGroup.bError THEN
				stError.ErrorId := fbBuildGroup.nErrorId;
				nStateA_Common := 99;
			ELSE
				IF stGCodeRef.pCurrentTool > 0 THEN
					IF (stGCodeRef.aToolTable[stGCodeRef.sNciToPlc.Tool].bIsInAction1 OR
						stGCodeRef.aToolTable[stGCodeRef.sNciToPlc.Tool].bIsInAction2 OR
						stGCodeRef.aToolTable[stGCodeRef.sNciToPlc.Tool].bIsInAction3) THEN
						nStateA_Common := 8;
					ELSE
						nStateA_Common := 9;
					END_IF
				ELSE
					nStateA_Common := 9;
				END_IF
			END_IF
			fbBuildGroup(stGCodeRef:= stGCodeRef, bExecute:= FALSE);
		END_IF
		
	8:	//letze PrintAction wieder starten (fall während des Prints unterbrochen)
		fbRestartPrintAct(stGCodeRef:= stGCodeRef, bExecute:= TRUE);
		IF NOT fbRestartPrintAct.bBusy THEN
			IF fbRestartPrintAct.bError THEN
				stError.ErrorId := fbRestartPrintAct.nErrorId;
				nStateA_Common := 99;
			ELSE
				nStateA_Common := 9;
			END_IF
			fbRestartPrintAct(stGCodeRef := stGCodeRef, bExecute:= FALSE);
		END_IF
		
	9:	//Interpreter starten
		fbItpStepOnAfterEStopEx(bExecute:= TRUE, sNciToPlc:= GCode.stGCodeRef.sNciToPlc);
		IF NOT fbItpStepOnAfterEStopEx.bBusy THEN
			IF fbItpStepOnAfterEStopEx.bErr THEN
				nStateA_Common := 99;
			ELSE
				nStateA_Common := 10;
			END_IF
			fbItpStepOnAfterEStopEx(bExecute:= FALSE, sNciToPlc:= GCode.stGCodeRef.sNciToPlc);
		END_IF
		
	10:	//SingleBlock-Mode verlassen
		fbItpSingleBlock(bExecuteModeChange:= TRUE,	nMode:= E_ItpSingleBlockMode.ItpSingleBlockOff, sNciToPlc:= GCode.stGCodeRef.sNciToPlc);
		IF NOT fbItpSingleBlock.bBusy THEN
			IF fbItpSingleBlock.bErr THEN
				nStateA_Common := 99;
			ELSE
				IF pHighVoltTray > 0 THEN
					//Strom-Überwachung wieder einschalten
					pHighVoltTray^.M_CurrentMonitoring(TRUE);
				END_IF				
				nStateA_Common := 80;
			END_IF
			fbItpSingleBlock(bExecuteModeChange:= FALSE, sNciToPlc:= GCode.stGCodeRef.sNciToPlc);
		END_IF		
END_CASE
END_ACTION

ACTION A_Init:
stError.POUState := nStateA_Common;

CASE nStateA_Common OF
	0:	//Checken, ob NCI vorhanden ist durch überprüfen des Mappings zur NCI
		IF F_GetMappingStatus(ADR(GCode.stGCodeRef.sNciToPlc),SIZEOF(GCode.stGCodeRef.sNciToPlc)) = EPlcMappingStatus.MS_Mapped THEN
			IF ItpGetStateInterpreter(GCode.stGCodeRef.sNciToPlc) > 0 THEN
				nStateA_Common := 2;
			END_IF
			bNciAvailable := TRUE;
		ELSE
			nStateA_Common := 81;	//NCI nicht verfügbar
		END_IF

		
	(*1:	//Berechnung der totalen Bahnlänge aktivieren
		dwAdsValue := 1;
		fbAdsWrite(PORT:= 501, IDXGRP:= 16#3000 + ItpGetGroupId(GCode.stGCodeRef.sNciToPlc), IDXOFFS:= 16#508, LEN:= SIZEOF(dwAdsValue), SRCADDR:=ADR(dwAdsValue), WRITE:= TRUE);
		IF NOT fbAdsWrite.BUSY THEN
			IF fbAdsWrite.ERR THEN
				stError.ErrorId := UDINT_TO_UINT(fbAdsWrite.ERRID);
				nStateA_Common := 99;
			END_IF
			fbAdsWrite(WRITE:= FALSE);
			nStateA_Common := 2;
		END_IF*)

	2:	//Aktiviere das Lesen der akt. wirkenden Interpolationsregeln, Nullp.verschiebungen & Rotation
		dwAdsValue := 1;
		fbAdsWrite(PORT:= 501, IDXGRP:= 16#2000 + ItpGetChannelId(GCode.stGCodeRef.sNciToPlc), IDXOFFS:= 16#53, LEN:= SIZEOF(dwAdsValue), SRCADDR:=ADR(dwAdsValue), WRITE:= TRUE);
		IF NOT fbAdsWrite.BUSY THEN
			IF fbAdsWrite.ERR THEN
				stError.ErrorId := UDINT_TO_UINT(fbAdsWrite.ERRID);
				nStateA_Common := 99;
			END_IF
			fbAdsWrite(WRITE:= FALSE);
			nStateA_Common := 3;
		END_IF

	3:	//Konfiguration zykl. Kanalinterface (frei konfigurierbaren "DoubleParams[0..3])
		fbItpSetCyclLrealOffs(bExecute:= TRUE , //nIndexOffsetParam1:= 16#522, (*Bahnrestweg (verbleibende Bogenlänge) auf dem aktuellen Bahnsegment*)
												//nIndexOffsetParam2:= 16#502, (*aktuelle Bahnsollgeschwindigkeit*)
												//nIndexOffsetParam3:= 16#509, (*Segmentübergang*)
												nIndexOffsetParam1:= 16#523, (*programmierte Geschwindigkeit des aktuellen Segments*)
												sNciToPlc:= GCode.stGCodeRef.sNciToPlc);

												
		IF NOT fbItpSetCyclLrealOffs.bBusy THEN
			nStateA_Common := 4;
			IF fbItpSetCyclLrealOffs.bErr THEN
				stError.ErrorId := UDINT_TO_UINT(fbItpSetCyclLrealOffs.nErrId);
				nStateA_Common := 99;
			END_IF
			fbItpSetCyclLrealOffs(bExecute:= FALSE, sNciToPlc:= GCode.stGCodeRef.sNciToPlc);
		END_IF
		
	4:	//Konfiguration zykl. Kanalinterface (frei konfigurierbaren "UdintParams[0..3])
		fbItpSetCyclUdintOffs(bExecute:= TRUE,	nIndexOffsetParam1:= 16#05, //SAF-Gruppenstatus (main state)
												sNciToPlc:= GCode.stGCodeRef.sNciToPlc);
		IF NOT fbItpSetCyclUdintOffs.bBusy THEN
			nStateA_Common := 5;
			IF fbItpSetCyclUdintOffs.bErr THEN
				stError.ErrorId := UDINT_TO_UINT(fbItpSetCyclUdintOffs.nErrId);
				nStateA_Common := 99;
			END_IF
			fbItpSetCyclUdintOffs(bExecute:= FALSE, sNciToPlc:= GCode.stGCodeRef.sNciToPlc);
		END_IF
		
	5:	//Q1-Achse einschalten (virtuell Achse)
		fbMcPower(Axis:= AxisRefQ1, Enable:= TRUE, Enable_Positive:= TRUE, Enable_Negative:= TRUE, Override:= 100);
		IF fbMcPower.Error THEN	 //Error bei Ausführung
			stError.ErrorId := UDINT_TO_UINT(fbMcPower.ErrorID);
			fbMcPower(Axis:= AxisRefQ1, Enable:= FALSE);
			nStateA_Common := 99;
		ELSE
			nStateA_Common := 6;
		END_IF
		
	6:	//Interpreter zurücksetzen
		fbItpResetEx2(bExecute:= TRUE, sNciToPlc:= GCode.stGCodeRef.sNciToPlc);
		IF NOT fbItpResetEx2.bBusy THEN
			IF fbItpResetEx2.bErr THEN
				stError.ErrorId := UDINT_TO_UINT(fbItpResetEx2.nErrId);
				nStateA_Common := 99;
			ELSE
				//ActionList initialisieren
				F_CreateLinkedListHnd(ADR(aNodes), SIZEOF(aNodes), hList);
				nStateA_Common := 80;				
			END_IF
			fbItpResetEx2(bExecute:= FALSE, sNciToPlc:= GCode.stGCodeRef.sNciToPlc);
		END_IF
		
END_CASE

IF nStateA_Common = 99 THEN
	stError.POUAction := E_POUACT.POUACT_A_Init;
	fbErrorList.M_Add(stError);
END_IF
END_ACTION

ACTION A_Load:
stError.POUState := nStateA_Common;

CASE nStateA_Common OF
	0:	//Interpreter zurücksetzen
		fbItpResetEx2(bExecute:= TRUE, sNciToPlc:= GCode.stGCodeRef.sNciToPlc);
		IF NOT fbItpResetEx2.bBusy THEN
			IF fbItpResetEx2.bErr THEN
				stError.ErrorId := UDINT_TO_UINT(fbItpResetEx2.nErrId);
				nStateA_Common := 99;
			ELSE
				nProgress := 0;
				nStateA_Common := 1;
			END_IF
			fbItpResetEx2(bExecute:= FALSE, sNciToPlc:= GCode.stGCodeRef.sNciToPlc);
		END_IF

	1:	//SingleBlock Mode ausschalten (falls durch Abbruch oder Fehler noch aktiv)
		fbItpSingleBlock(bExecuteModeChange:= TRUE,	nMode:= Tc2_NCI.E_ItpSingleBlockMode.ItpSingleBlockOff,
						bTriggerNext:= FALSE, sNciToPlc:= GCode.stGCodeRef.sNciToPlc);
		IF NOT fbItpSingleBlock.bBusy THEN
			IF fbItpSingleBlock.bErr THEN
				stError.ErrorId := UDINT_TO_UINT(fbItpSingleBlock.nErrId);
				nStateA_Common := 99;
			ELSE
				nStateA_Common := 2;
			END_IF
			fbItpSingleBlock(bExecuteModeChange:= FALSE, bTriggerNext:= FALSE, sNciToPlc:= GCode.stGCodeRef.sNciToPlc);
		END_IF
		
		(*
	2:  Der Funktionsbaustein ItpEnableDefaultGCode ermöglicht es, aus der SPS einen vom Anwender definierten G-Code vor dem Start jedes NC-Programms auszuführen. 
		Das Defaultprogramm wird beim Start des eigentlichen NC-Programms vor dem geladenen Programm ausgeführt.
		Mit diesem Funktionsbaustein ist es zum Beispiel möglich, das Koordinatensystem für alle auszuführenden NC-Programme zu drehen.
		Der Standard-G-Code muss als „DefaultGCode<Channel-Number>.def“ im TwinCAT\CNC Verzeichnis gespeichert werden
		fbItpEnableDefaultGCode(bUseDefaultGCode:= TRUE, bExecute:= TRUE, sNciToPlc:= GCode.stGCodeRef.sNciToPlc, tTimeOut:= T#20S);
		IF NOT fbItpEnableDefaultGCode.bBusy THEN
			IF fbItpEnableDefaultGCode.bErr THEN
				stError.ErrorId := UDINT_TO_UINT(fbItpEnableDefaultGCode.nErrId);
				nStateA_Common := 99;
			ELSE
				nStateA_Common := 3;	
			END_IF
			fbItpEnableDefaultGCode(bExecute:= FALSE, sNciToPlc:= GCode.stGCodeRef.sNciToPlc);
		END_IF*)
		
	2:	//GCode-File laden (ab hier erfolgt Syntaxüberprüfung)
		//Langes Timeout bei große Dateien erforderlich
		fbItpLoadProgEx(bExecute:= TRUE, sNciToPlc:= GCode.stGCodeRef.sNciToPlc, sPrg:= sGCodeFile ,nLength:= INT_TO_UINT(LEN(sGCodeFile)),tTimeOut:= T#120S);
		IF NOT fbItpLoadProgEx.bBusy THEN
			IF fbItpLoadProgEx.bErr THEN
				stError.ErrorId := UDINT_TO_UINT(fbItpLoadProgEx.nErrId);
				nStateA_Common := 99;
			ELSE
				nStateA_Common := 3;	
			END_IF
			fbItpLoadProgEx(bExecute:= FALSE, sNciToPlc:= GCode.stGCodeRef.sNciToPlc);
		END_IF
		
	3:	//Dateigröße ermitteln
		fbEnumFindFileEntry(sPathName:= sGCodeFile,	eCmd:= E_EnumCmdType.eEnumCmd_First, bExecute:= TRUE, stFindFile=> stFindFile);
		IF NOT fbEnumFindFileEntry.bBusy THEN
			IF fbEnumFindFileEntry.bError THEN
				nStateA_Common := 99;
			ELSE
				nStateA_Common := 4;
			END_IF
			fbEnumFindFileEntry(sPathName:= sGCodeFile,	eCmd:= E_EnumCmdType.eEnumCmd_First, bExecute:= FALSE);
		END_IF
		
	4:	fbEnumFindFileEntry(eCmd:= E_EnumCmdType.eEnumCmd_Abort, bExecute:= TRUE);
		IF NOT fbEnumFindFileEntry.bBusy THEN
			IF fbEnumFindFileEntry.bError THEN
				nStateA_Common := 99;
			ELSE
				nStateA_Common := 80;
			END_IF
			fbEnumFindFileEntry(sPathName:= sGCodeFile,	eCmd:= E_EnumCmdType.eEnumCmd_First, bExecute:= FALSE);
		END_IF
		
END_CASE

IF nStateA_Common = 99 THEN
	stError.POUAction := E_POUACT.POUACT_A_Load;
	fbErrorList.M_Add(stError);
END_IF
END_ACTION

ACTION A_Pause:
stError.POUState := nStateA_Common;

IF stGCodeRef.sNciToPlc.IntParams[0] = E_SAF_State.Control AND bLockPause THEN
	bLockPause := FALSE;
END_IF

//Falls noch eine FastMFunc anliegt, verhindern, dass SingleBlock aktiviert wird
fbFastMFunc(stGCodeRef:= stGCodeRef, bStop:= FALSE);
IF fbFastMFunc.bBusy THEN
	fbFastMFunc(stGCodeRef:= stGCodeRef, bStop:= FALSE);
	bLockPause := TRUE;
	RETURN;
END_IF

//Falls noch eine HSKMFunc anliegt, verhindern, dass SingleBlock aktiviert wird
//Falls eine pausierbare HSKMFunc anliegt, dann diese in Pause versetzen
//In diesem Falls bleibt die HSKMFunc noch aktiv und der GCode-Interpreter wird nicht in Singleblock versetzt
//wichtig beim Continue -> dort wird einfach die HSKMFunc wieder aktiv

fbHskMFunc(stGCodeRef:= stGCodeRef, pXDrive:= pXDrive, pYDrive:= pYDrive, bStop:= FALSE, bPause:= TRUE, bContinue:= FALSE);
IF fbHskMFunc.bBusy THEN
	fbHskMFunc(stGCodeRef:= stGCodeRef, pXDrive:= pXDrive, pYDrive:= pYDrive, bStop:= FALSE, bPause:= TRUE, bContinue:= FALSE);
	IF fbHskMFunc.bIsInPause THEN
		bLockPause := FALSE;
		nStateA_Common := 80;
	ELSE
		bLockPause := TRUE;	
	END_IF
	RETURN;
END_IF

IF stInfo.nNciState = Tc2_NCI.NCI_INTERPRETER_READY THEN
	nStateA_Common := 80;
	RETURN;
END_IF

CASE nStateA_Common OF
	0:			
		IF bLockPause THEN
			RETURN;
		END_IF
		
		//In Singleblock setzen, erst wenn SAF-State wieder Run
		IF stGCodeRef.sNciToPlc.IntParams[0] = E_SAF_State.Control THEN
			RETURN;
		END_IF
		
		fbItpSingleBlock(bExecuteModeChange:= TRUE,	nMode:= E_ItpSingleBlockMode.ItpSingleBlockNck, bTriggerNext:= FALSE, sNciToPlc:= GCode.stGCodeRef.sNciToPlc);
		IF NOT fbItpSingleBlock.bBusy THEN
			IF fbItpSingleBlock.bErr THEN
				stError.ErrorId := UDINT_TO_UINT(fbItpSingleBlock.nErrId);
				nStateA_Common := 99;
			ELSE
				nStateA_Common := 1;	
			END_IF
			fbItpSingleBlock(bExecuteModeChange:= FALSE, sNciToPlc:= GCode.stGCodeRef.sNciToPlc);
		END_IF
		
	1:	//letzer Befehl abgearbeitet?
		IF NOT (stGCodeRef.pHead^.P_pXDrive^.P_bIsMoving OR stGCodeRef.pHead^.P_pYDrive^.P_bIsMoving) THEN	//Bewegung noch aktiv
			nStateA_Common := 2;
			//Aktive Tool eine MES-Cartridge? -> StopPrintAction überspringen
			IF stGCodeRef.pCurrentTool^.P_eObjectType = E_ObjectType.OBJECTTYPE_CartDispenser OR
										stGCodeRef.pCurrentTool^.P_eObjectType = E_ObjectType.OBJECTTYPE_CartDispStirrer THEN
				pMesCartDisp := stGCodeRef.pCurrentTool;
				IF pMesCartDisp^.P_bIsMESTool THEN
					RETURN;
				END_IF
			END_IF
			//Print-Action stoppen
			fbFastMFunc.M_StopPrintAction(stGCodeRef.pCurrentTool,0);
		END_IF
		
	2:	//Interpreter stoppen
		fbItpEStopEx(sNciToPlc:= GCode.stGCodeRef.sNciToPlc, bExecute:= TRUE);
		IF NOT fbItpEStopEx.bBusy THEN
			IF fbItpEStopEx.bErr THEN
				stError.ErrorId := UDINT_TO_UINT(fbItpEStopEx.nErrId);
				nStateA_Common := 99;
			ELSE
				nStateA_Common := 3;
			END_IF
			fbItpEStopEx(sNciToPlc:= GCode.stGCodeRef.sNciToPlc, bExecute:= FALSE);
		END_IF
		
	3:	//Warten bis SAF = Control
		IF stGCodeRef.sNciToPlc.IntParams[0] = E_SAF_State.Control THEN
			nStateA_Common := 4;
		END_IF
		
	4:	//Gruppe auflösen
		stMethResult := M_ClearGroup(TRUE);
		IF NOT stMethResult.bBusy THEN
			IF stMethResult.bError THEN
				stError.ErrorId := stMethResult.nErrorId;
				nStateA_Common := 99;
			ELSE
				//Aktuelle Position merken zum zurückfahren
				//Wenn pCurrentTool noch nicht gesetzt wurde, weil die Hsk-Func SelectTool noch nicht ausgeführt wurde, dann
				//braucht im Grunde nicht zurückgefahren werden
				IF stGCodeRef.pCurrentTool > 0 THEN
					//wird in A_Continue benötigt
					stCurrentPos := stGCodeRef.pCurrentTool^.P_stCurrentPosTotal;
				END_IF
				nStateA_Common := 5;
				IF stGCodeRef.pCurrentTool^.P_eObjectType = E_ObjectType.OBJECTTYPE_CartDispenser OR
										stGCodeRef.pCurrentTool^.P_eObjectType = E_ObjectType.OBJECTTYPE_CartDispStirrer THEN
					pMesCartDisp := stGCodeRef.pCurrentTool;
					IF pMesCartDisp^.P_bIsMESTool THEN
						nStateA_Common := 80;
					END_IF
				END_IF				
			END_IF
		END_IF
		
	5:	//MoveZ free
		stActionDataMoveZ.eAction := E_Action.ACTION_MoveZ;
		stActionDataMoveZ.aParams[1] := E_MoveMode.MODE_Free;
		stActionDataMoveZ.aParams[3]:= -1; //MaxSpeed
		stError.ErrorId := stGCodeRef.pCurrentTool^.M_ExeAction(stActionDataMoveZ);
		
		IF  stError.ErrorId > 0 THEN
			nStateA_Common := 99;
		ELSE
			nStateA_Common := 6;
		END_IF		
	
	6:	//MoveZ ready?
		IF NOT stGCodeRef.pCurrentTool^.M_GetActionBusy(E_Action.ACTION_MoveZ) THEN
			IF stGCodeRef.pCurrentTool^.P_bError THEN
				stError.ErrorId := stGCodeRef.pCurrentTool^.P_nErrorId;
				nStateA_Common := 99;
			ELSE
				nStateA_Common := 80;
			END_IF
		END_IF	
END_CASE

IF nStateA_Common = 99 THEN
	stError.POUAction := E_POUACT.POUACT_A_Pause;
	fbErrorList.M_Add(stError);
END_IF
END_ACTION

ACTION A_Reset:
stError.POUState := nStateA_Common;

CASE nStateA_Common OF
	0:	//Interpreter zurücksetzen
		fbItpResetEx2(bExecute:= TRUE, sNciToPlc:= GCode.stGCodeRef.sNciToPlc);
		IF NOT fbItpResetEx2.bBusy THEN
			IF fbItpResetEx2.bErr THEN
				stError.ErrorId := UDINT_TO_UINT(fbItpResetEx2.nErrId);
				nStateA_Common := 99;
			ELSE
				nStateA_Common := 1;
			END_IF
			fbItpResetEx2(bExecute:= FALSE, sNciToPlc:= GCode.stGCodeRef.sNciToPlc);
		END_IF
		
	1:	//Interpolationsgruppe löschen
		stMethResult := M_ClearGroup(TRUE);
		IF NOT stMethResult.bBusy THEN
			IF stMethResult.bError THEN
				stError.ErrorId := stMethResult.nErrorId;
				nStateA_Common := 99;
			ELSE
				nStateA_Common := 80;
				bError := FALSE;
				bMoveActionsLocked := FALSE;
			END_IF
		END_IF

END_CASE

IF nStateA_Common = 99 THEN
	stError.POUAction := E_POUACT.POUACT_A_Reset;
	fbErrorList.M_Add(stError);	
END_IF
END_ACTION

ACTION A_Run:
stError.POUState := nStateA_Common;
stInfo.nNciState := ItpGetStateInterpreter(stGCodeRef.sNciToPlc);
ItpSetOverridePercent(stGCodeRef.lrNcOverride,stGCodeRef.sPlcToNci);

CASE nStateA_Common OF
	0:	//*****Running*****
		IF bStop THEN
			nStateA_Common := 5;
			//nStateA_CommonNext := 80;
		ELSE
			CASE stInfo.nNciState OF
				Tc2_NCI.NCI_INTERPRETER_IDLE:
					nStateA_Common := 10;
					nStateA_CommonNext := 80;
				Tc2_NCI.NCI_INTERPRETER_READY:
					nStateA_Common := 10;
					nStateA_CommonNext := 80;
				Tc2_NCI.NCI_INTERPRETER_RUNNING:
					//FastMFunc auswerten
					fbFastMFunc(stGCodeRef:= stGCodeRef,bStop:= FALSE);
					IF fbFastMFunc.bError THEN
						stError.ErrorId := fbFastMFunc.nErrorId;
						nStateA_Common := 10;
						nStateA_CommonNext := 99;
					ELSE
						//HskMFunc auswerten
						fbHskMFunc(stGCodeRef:= stGCodeRef, pXDrive:= pXDrive, pYDrive:= pYDrive, bStop:= FALSE);
						IF fbHskMFunc.bError THEN
							nStateA_Common := 10;
							nStateA_CommonNext := 99;
						ELSIF fbHskMFunc.bCanceled THEN
							nStateA_Common := 10;
							nStateA_CommonNext := 80;
						ELSE
							//Stromüberwachung
							IF pHighVoltTray > 0 THEN
								IF pHighVoltTray^.P_bPwrCutOffTriggered THEN
									nStateA_Common := 5;
								END_IF
							END_IF
							//Sobald das aktive Tool in Error geht, Abbrechen!
							IF stGCodeRef.pCurrentTool > 0 AND_THEN stGCodeRef.pCurrentTool^.P_bError THEN
								nStateA_Common := 5;
							END_IF
						END_IF
					END_IF
					
				Tc2_NCI.NCI_INTERPRETER_SINGLESTOP:
					;
				Tc2_NCI.NCI_INTERPRETER_WAITFUNC:
					;
				Tc2_NCI.NCI_INTERPRETER_FAULT:
					stError.ErrorId := UDINT_TO_UINT(ItpGetError(stGCodeRef.sNciToPlc));
					nStateA_Common := 10;
					nStateA_CommonNext := 99;
				Tc2_NCI.NCI_INTERPRETER_ABORTED:
					stError.ErrorId := UDINT_TO_UINT(ItpGetError(stGCodeRef.sNciToPlc));
					nStateA_Common := 10;
					nStateA_CommonNext := 99;
				Tc2_NCI.NCI_INTERPRETER_FLUSHBUFFERS:
					nStateA_Common := 10;
					nStateA_CommonNext := 99;
			END_CASE
		END_IF
		
	5:	//Stoppen
		//Sicherstellen, dass FastMFunc und HskMFunc beendet wurden bzw diese beenden
		//Durch StopAll werden die Devices bzw. die ComplexActions gestoppt.
		//Durch StopAction müssen diese noch gestoppt werden
		//Die Methoden erhalten einen Eingang "bStop"
		nStateA_Common := 10;
		nStateA_CommonNext := 80;
		IF fbFastMFunc.bBusy THEN
			fbFastMFunc(stGCodeRef:= stGCodeRef, bStop:= TRUE);
			nStateA_Common := 5;
		END_IF
		
		IF fbHskMFunc.bBusy THEN
			fbHskMFunc(stGCodeRef:= stGCodeRef, pXDrive:= pXDrive, pYDrive:= pYDrive, bStop:= TRUE, bPause:= FALSE, bContinue:= FALSE);
			nStateA_Common := 5;
		END_IF
		
		IF NOT (fbFastMFunc.bBusy OR fbHskMFunc.bBusy) THEN
			fbFastMFunc.M_StopPrintAction(stGCodeRef.pCurrentTool,0);
		END_IF
	
